LIN {X 0,Y 191.055,Z 844.267,A -85,B 0,C 180,E1 -30758.492,E2 -30758.492} C_VEL
LIN {X 0,Y 183.715,Z 843.37,A -85,B 0,C 180,E1 -30762.24,E2 -30762.24} C_VEL
LIN {X 0,Y 177.701,Z 841.067,A -85,B 0,C 180,E1 -30766.319,E2 -30766.319} C_VEL
LIN {X 0,Y 173.965,Z 838.465,A -85,B 0,C 180,E1 -30769.56,E2 -30769.56} C_VEL
LIN {X 0,Y 170.368,Z 833.668,A -85,B 0,C 180,E1 -30774.1,E2 -30774.1} C_VEL
LIN {X 0,Y 168.598,Z 829.177,A -85,B 0,C 180,E1 -30777.618,E2 -30777.618} C_VEL
LIN {X 0,Y 167.407,Z 822.526,A -85,B 0,C 180,E1 -30781.797,E2 -30781.797} C_VEL
LIN {X 0,Y 167.191,Z 815.652,A -85,B 0,C 180,E1 -30785.408,E2 -30785.408} C_VEL
LIN {X 0,Y 167.388,Z 808.865,A -85,B 0,C 180,E1 -30788.421,E2 -30788.421} C_VEL
LIN {X 0,Y 167.699,Z 800.631,A -85,B 0,C 180,E1 -30791.442,E2 -30791.442} C_VEL
LIN {X 0,Y 167.988,Z 791.47,A -85,B 0,C 180,E1 -30794.179,E2 -30794.179} C_VEL
LIN {X 0,Y 168.367,Z 782.647,A -85,B 0,C 180,E1 -30796.399,E2 -30796.399} C_VEL
LIN {X 0,Y 168.769,Z 772.895,A -85,B 0,C 180,E1 -30798.447,E2 -30798.447} C_VEL
LIN {X 0,Y 169.197,Z 762.216,A -85,B 0,C 180,E1 -30800.285,E2 -30800.285} C_VEL
LIN {X 0,Y 169.704,Z 751.249,A -85,B 0,C 180,E1 -30801.805,E2 -30801.805} C_VEL
LIN {X 0,Y 170.027,Z 740.5,A -85,B 0,C 180,E1 -30802.958,E2 -30802.958} C_VEL
LIN {X 0,Y 171.114,Z 700.591,A -85,B 0,C 180,E1 -30806.113,E2 -30806.113} C_VEL
LIN {X 0,Y 171.929,Z 668.174,A -85,B 0,C 180,E1 -30808.506,E2 -30808.506} C_VEL
LIN {X 0,Y 169.464,Z 639.672,A -85,B 0,C 180,E1 -30810.518,E2 -30810.518} C_VEL
LIN {X 0,Y 169.295,Z 636.336,A -85,B 0,C 180,E1 -30810.797,E2 -30810.797} C_VEL
LIN {X 0,Y 168.528,Z 636.419,A -85,B 0,C 180,E1 -30817.843,E2 -30817.843} C_VEL
LIN {X 0,Y 168.51,Z 636.427,A -85,B 0,C 180,E1 -30821.686,E2 -30821.686} C_VEL
LIN {X 0,Y 168.522,Z 636.419,A -85,B 0,C 180,E1 -30825.041,E2 -30825.041} C_VEL
LIN {X 0,Y 168.51,Z 636.425,A -85,B 0,C 180,E1 -30828.434,E2 -30828.434} C_VEL
LIN {X 0,Y 168.485,Z 636.43,A -85,B 0,C 180,E1 -30832.174,E2 -30832.174} C_VEL
LIN {X 0,Y 168.489,Z 636.423,A -85,B 0,C 180,E1 -30837.286,E2 -30837.286} C_VEL
LIN {X 0,Y 168.541,Z 636.422,A -85,B 0,C 180,E1 -30840.777,E2 -30840.777} C_VEL
LIN {X 0,Y 168.602,Z 636.409,A -85,B 0,C 180,E1 -30846.058,E2 -30846.058} C_VEL
LIN {X 0,Y 168.727,Z 636.397,A -85,B 0,C 180,E1 -30852.705,E2 -30852.705} C_VEL
LIN {X 0,Y 168.823,Z 636.386,A -85,B 0,C 180,E1 -30858.027,E2 -30858.027} C_VEL
LIN {X 0,Y 169.224,Z 636.335,A -85,B 0,C 180,E1 -30863.403,E2 -30863.403} C_VEL
LIN {X 0,Y 169.389,Z 636.314,A -85,B 0,C 180,E1 -30867.63,E2 -30867.63} C_VEL
LIN {X 0,Y 169.471,Z 636.309,A -85,B 0,C 180,E1 -30870,E2 -30870} C_VEL
LIN {X 0,Y 169.237,Z 636.327,A -85,B 0,C 180,E1 -30874.748,E2 -30874.748} C_VEL
LIN {X 0,Y 169.13,Z 636.346,A -85,B 0,C 180,E1 -30877.137,E2 -30877.137} C_VEL
LIN {X 0,Y 168.823,Z 636.386,A -85,B 0,C 180,E1 -30881.972,E2 -30881.972} C_VEL
LIN {X 0,Y 168.726,Z 636.397,A -85,B 0,C 180,E1 -30887.294,E2 -30887.294} C_VEL
LIN {X 0,Y 168.6,Z 636.409,A -85,B 0,C 180,E1 -30893.941,E2 -30893.941} C_VEL
LIN {X 0,Y 168.543,Z 636.422,A -85,B 0,C 180,E1 -30899.224,E2 -30899.224} C_VEL
LIN {X 0,Y 168.513,Z 636.42,A -85,B 0,C 180,E1 -30903.767,E2 -30903.767} C_VEL
LIN {X 0,Y 168.501,Z 636.428,A -85,B 0,C 180,E1 -30908.574,E2 -30908.574} C_VEL
LIN {X 0,Y 168.51,Z 636.425,A -85,B 0,C 180,E1 -30911.687,E2 -30911.687} C_VEL
LIN {X 0,Y 168.52,Z 636.42,A -85,B 0,C 180,E1 -30915.043,E2 -30915.043} C_VEL
LIN {X 0,Y 168.51,Z 636.427,A -85,B 0,C 180,E1 -30918.435,E2 -30918.435} C_VEL
LIN {X 0,Y 168.494,Z 636.423,A -85,B 0,C 180,E1 -30922.171,E2 -30922.171} C_VEL
LIN {X 0,Y 168.503,Z 636.426,A -85,B 0,C 180,E1 -30927.291,E2 -30927.291} C_VEL
LIN {X 0,Y 168.542,Z 636.414,A -85,B 0,C 180,E1 -30932.798,E2 -30932.798} C_VEL
LIN {X 0,Y 168.553,Z 636.423,A -85,B 0,C 180,E1 -30938.038,E2 -30938.038} C_VEL
LIN {X 0,Y 168.728,Z 636.39,A -85,B 0,C 180,E1 -30943.108,E2 -30943.108} C_VEL
LIN {X 0,Y 168.777,Z 636.395,A -85,B 0,C 180,E1 -30948.025,E2 -30948.025} C_VEL
LIN {X 0,Y 169.227,Z 636.329,A -85,B 0,C 180,E1 -30953.4,E2 -30953.4} C_VEL
LIN {X 0,Y 169.395,Z 636.317,A -85,B 0,C 180,E1 -30957.631,E2 -30957.631} C_VEL
LIN {X 0,Y 169.471,Z 636.305,A -85,B 0,C 180,E1 -30960.001,E2 -30960.001} C_VEL
LIN {X 0,Y 169.24,Z 636.333,A -85,B 0,C 180,E1 -30964.749,E2 -30964.749} C_VEL
LIN {X 0,Y 169.131,Z 636.349,A -85,B 0,C 180,E1 -30967.138,E2 -30967.138} C_VEL
LIN {X 0,Y 168.769,Z 636.388,A -85,B 0,C 180,E1 -30971.977,E2 -30971.977} C_VEL
LIN {X 0,Y 168.652,Z 636.408,A -85,B 0,C 180,E1 -30977.21,E2 -30977.21} C_VEL
LIN {X 0,Y 168.551,Z 636.418,A -85,B 0,C 180,E1 -30983.902,E2 -30983.902} C_VEL
LIN {X 0,Y 168.543,Z 636.42,A -85,B 0,C 180,E1 -30989.223,E2 -30989.223} C_VEL
LIN {X 0,Y 168.47,Z 636.428,A -85,B 0,C 180,E1 -30993.744,E2 -30993.744} C_VEL
LIN {X 0,Y 168.474,Z 636.429,A -85,B 0,C 180,E1 -30998.583,E2 -30998.583} C_VEL
LIN {X 0,Y 168.459,Z 636.425,A -85,B 0,C 180,E1 -31001.704,E2 -31001.704} C_VEL
LIN {X 0,Y 168.461,Z 636.432,A -85,B 0,C 180,E1 -31005.022,E2 -31005.022} C_VEL
LIN {X 0,Y 168.465,Z 636.43,A -85,B 0,C 180,E1 -31008.453,E2 -31008.453} C_VEL
LIN {X 0,Y 168.479,Z 636.425,A -85,B 0,C 180,E1 -31012.179,E2 -31012.179} C_VEL
LIN {X 0,Y 168.51,Z 636.426,A -85,B 0,C 180,E1 -31017.292,E2 -31017.292} C_VEL
LIN {X 0,Y 168.863,Z 636.379,A -85,B 0,C 180,E1 -31022.853,E2 -31022.853} C_VEL
LIN {X 0,Y 169.387,Z 636.322,A -85,B 0,C 180,E1 -31025.575,E2 -31025.575} C_VEL
LIN {X 0,Y 169.125,Z 636.516,A -85,B 0,C 180,E1 -31026.992,E2 -31026.992} C_VEL
LIN {X 0,Y 168.664,Z 639.876,A -85,B 0,C 180,E1 -31028.932,E2 -31028.932} C_VEL
LIN {X 0,Y 169.406,Z 663.952,A -85,B 0,C 180,E1 -31030.685,E2 -31030.685} C_VEL
LIN {X 0,Y 171.642,Z 691.866,A -85,B 0,C 180,E1 -31032.65,E2 -31032.65} C_VEL
LIN {X 0,Y 170.5,Z 744.148,A -85,B 0,C 180,E1 -31036.64,E2 -31036.64} C_VEL
LIN {X 0,Y 170.205,Z 756.052,A -85,B 0,C 180,E1 -31037.825,E2 -31037.825} C_VEL
LIN {X 0,Y 169.892,Z 767.351,A -85,B 0,C 180,E1 -31039.308,E2 -31039.308} C_VEL
LIN {X 0,Y 169.553,Z 776.429,A -85,B 0,C 180,E1 -31040.789,E2 -31040.789} C_VEL
LIN {X 0,Y 169.206,Z 786.88,A -85,B 0,C 180,E1 -31042.867,E2 -31042.867} C_VEL
LIN {X 0,Y 168.997,Z 795.616,A -85,B 0,C 180,E1 -31044.947,E2 -31044.947} C_VEL
LIN {X 0,Y 168.892,Z 803.11,A -85,B 0,C 180,E1 -31047.029,E2 -31047.029} C_VEL
LIN {X 0,Y 168.902,Z 810.469,A -85,B 0,C 180,E1 -31049.406,E2 -31049.406} C_VEL
LIN {X 0,Y 168.775,Z 818.031,A -85,B 0,C 180,E1 -31052.379,E2 -31052.379} C_VEL
LIN {X 0,Y 168.286,Z 825.103,A -85,B 0,C 180,E1 -31055.973,E2 -31055.973} C_VEL
LIN {X 0,Y 168,Z 830.869,A -85,B 0,C 180,E1 -31059.601,E2 -31059.601} C_VEL
LIN {X 0,Y 168.608,Z 835.707,A -85,B 0,C 180,E1 -31063.208,E2 -31063.208} C_VEL
LIN {X 0,Y 170.819,Z 840.683,A -85,B 0,C 180,E1 -31067.911,E2 -31067.911} C_VEL
LIN {X 0,Y 173.542,Z 843.594,A -85,B 0,C 180,E1 -31071.301,E2 -31071.301} C_VEL
LIN {X 0,Y 178.333,Z 846.216,A -85,B 0,C 180,E1 -31075.598,E2 -31075.598} C_VEL
LIN {X 0,Y 184.426,Z 847.512,A -85,B 0,C 180,E1 -31079.587,E2 -31079.587} C_VEL
LIN {X 0,Y 187.854,Z 847.692,A -85,B 0,C 180,E1 -31081.468,E2 -31081.468} C_VEL
LIN {X 0,Y 195.715,Z 847.111,A -85,B 0,C 180,E1 -31084.934,E2 -31084.934} C_VEL
LIN {X 0,Y 205.771,Z 844.746,A -85,B 0,C 180,E1 -31088.471,E2 -31088.471} C_VEL
LIN {X 0,Y 216.568,Z 840.579,A -85,B 0,C 180,E1 -31091.532,E2 -31091.532} C_VEL
LIN {X 0,Y 224.354,Z 836.762,A -85,B 0,C 180,E1 -31093.382,E2 -31093.382} C_VEL
LIN {X 0,Y 232.555,Z 831.917,A -85,B 0,C 180,E1 -31095.058,E2 -31095.058} C_VEL
LIN {X 0,Y 241.045,Z 825.94,A -85,B 0,C 180,E1 -31096.592,E2 -31096.592} C_VEL
LIN {X 0,Y 248.373,Z 820.093,A -85,B 0,C 180,E1 -31097.756,E2 -31097.756} C_VEL
LIN {X 0,Y 257.164,Z 811.844,A -85,B 0,C 180,E1 -31098.992,E2 -31098.992} C_VEL
LIN {X 0,Y 264.177,Z 804.216,A -85,B 0,C 180,E1 -31099.877,E2 -31099.877} C_VEL
LIN {X 0,Y 263.17,Z 805.387,A -85,B 0,C 180,E1 -31100.012,E2 -31100.012} C_VEL
LIN {X 0,Y 257.968,Z 810.774,A -85,B 0,C 180,E1 -31099.94,E2 -31099.94} C_VEL
LIN {X 0,Y 253.897,Z 814.812,A -85,B 0,C 180,E1 -31099.733,E2 -31099.733} C_VEL
LIN {X 0,Y 245.545,Z 821.967,A -85,B 0,C 180,E1 -31099.109,E2 -31099.109} C_VEL
LIN {X 0,Y 241.416,Z 825.04,A -85,B 0,C 180,E1 -31098.602,E2 -31098.602} C_VEL
LIN {X 0,Y 233.412,Z 830.545,A -85,B 0,C 180,E1 -31097.326,E2 -31097.326} C_VEL
LIN {X 0,Y 224.856,Z 835.559,A -85,B 0,C 180,E1 -31095.764,E2 -31095.764} C_VEL
LIN {X 0,Y 216.603,Z 839.644,A -85,B 0,C 180,E1 -31094.049,E2 -31094.049} C_VEL
LIN {X 0,Y 208.795,Z 842.789,A -85,B 0,C 180,E1 -31092.14,E2 -31092.14} C_VEL
LIN {X 0,Y 201.117,Z 845.175,A -85,B 0,C 180,E1 -31089.985,E2 -31089.985} C_VEL
LIN {X 0,Y 194.363,Z 846.653,A -85,B 0,C 180,E1 -31087.782,E2 -31087.782} C_VEL
LIN {X 0,Y 185.778,Z 847.498,A -85,B 0,C 180,E1 -31084.441,E2 -31084.441} C_VEL
LIN {X 0,Y 178.316,Z 847.013,A -85,B 0,C 180,E1 -31080.708,E2 -31080.708} C_VEL
LIN {X 0,Y 172.018,Z 845.234,A -85,B 0,C 180,E1 -31076.61,E2 -31076.61} C_VEL
LIN {X 0,Y 167.071,Z 842.215,A -85,B 0,C 180,E1 -31072.169,E2 -31072.169} C_VEL
LIN {X 0,Y 164.258,Z 839.064,A -85,B 0,C 180,E1 -31068.653,E2 -31068.653} C_VEL
LIN {X 0,Y 162.431,Z 835.186,A -85,B 0,C 180,E1 -31064.996,E2 -31064.996} C_VEL
LIN {X 0,Y 161.476,Z 830.456,A -85,B 0,C 180,E1 -31061.257,E2 -31061.257} C_VEL
LIN {X 0,Y 161.73,Z 822.463,A -85,B 0,C 180,E1 -31056.215,E2 -31056.215} C_VEL
LIN {X 0,Y 162.123,Z 816.783,A -85,B 0,C 180,E1 -31053.287,E2 -31053.287} C_VEL
LIN {X 0,Y 162.247,Z 808.731,A -85,B 0,C 180,E1 -31050,E2 -31050} C_VEL
LIN {X 0,Y 162.202,Z 798.946,A -85,B 0,C 180,E1 -31046.845,E2 -31046.845} C_VEL
LIN {X 0,Y 162.351,Z 789.872,A -85,B 0,C 180,E1 -31044.43,E2 -31044.43} C_VEL
LIN {X 0,Y 162.561,Z 780.372,A -85,B 0,C 180,E1 -31042.321,E2 -31042.321} C_VEL
LIN {X 0,Y 162.988,Z 769.102,A -85,B 0,C 180,E1 -31040.274,E2 -31040.274} C_VEL
LIN {X 0,Y 163.288,Z 758.249,A -85,B 0,C 180,E1 -31038.714,E2 -31038.714} C_VEL
LIN {X 0,Y 163.548,Z 746.284,A -85,B 0,C 180,E1 -31037.4,E2 -31037.4} C_VEL
LIN {X 0,Y 164.158,Z 713.491,A -85,B 0,C 180,E1 -31034.692,E2 -31034.692} C_VEL
LIN {X 0,Y 164.481,Z 689.282,A -85,B 0,C 180,E1 -31032.777,E2 -31032.777} C_VEL
LIN {X 0,Y 161.917,Z 656.305,A -85,B 0,C 180,E1 -31030.339,E2 -31030.339} C_VEL
LIN {X 0,Y 161.586,Z 639.7,A -85,B 0,C 180,E1 -31029.046,E2 -31029.046} C_VEL
LIN {X 0,Y 161.826,Z 637.261,A -85,B 0,C 180,E1 -31027.578,E2 -31027.578} C_VEL
LIN {X 0,Y 162.227,Z 637.213,A -85,B 0,C 180,E1 -31025.056,E2 -31025.056} C_VEL
LIN {X 0,Y 161.479,Z 637.299,A -85,B 0,C 180,E1 -31018.633,E2 -31018.633} C_VEL
LIN {X 0,Y 161.427,Z 637.309,A -85,B 0,C 180,E1 -31015.531,E2 -31015.531} C_VEL
LIN {X 0,Y 161.43,Z 637.299,A -85,B 0,C 180,E1 -31011.355,E2 -31011.355} C_VEL
LIN {X 0,Y 161.383,Z 637.316,A -85,B 0,C 180,E1 -31006.018,E2 -31006.018} C_VEL
LIN {X 0,Y 161.386,Z 637.306,A -85,B 0,C 180,E1 -31000.62,E2 -31000.62} C_VEL
LIN {X 0,Y 161.414,Z 637.31,A -85,B 0,C 180,E1 -30997.411,E2 -30997.411} C_VEL
LIN {X 0,Y 161.405,Z 637.312,A -85,B 0,C 180,E1 -30994.345,E2 -30994.345} C_VEL
LIN {X 0,Y 161.471,Z 637.3,A -85,B 0,C 180,E1 -30989.822,E2 -30989.822} C_VEL
LIN {X 0,Y 161.488,Z 637.301,A -85,B 0,C 180,E1 -30984.376,E2 -30984.376} C_VEL
LIN {X 0,Y 161.487,Z 637.296,A -85,B 0,C 180,E1 -30980.304,E2 -30980.304} C_VEL
LIN {X 0,Y 161.615,Z 637.283,A -85,B 0,C 180,E1 -30975.073,E2 -30975.073} C_VEL
LIN {X 0,Y 161.838,Z 637.255,A -85,B 0,C 180,E1 -30969.97,E2 -30969.97} C_VEL
LIN {X 0,Y 162.186,Z 637.214,A -85,B 0,C 180,E1 -30966.632,E2 -30966.632} C_VEL
LIN {X 0,Y 162.354,Z 637.186,A -85,B 0,C 180,E1 -30962.473,E2 -30962.473} C_VEL
LIN {X 0,Y 162.439,Z 637.181,A -85,B 0,C 180,E1 -30960.001,E2 -30960.001} C_VEL
LIN {X 0,Y 162.19,Z 637.211,A -85,B 0,C 180,E1 -30955.046,E2 -30955.046} C_VEL
LIN {X 0,Y 162.059,Z 637.222,A -85,B 0,C 180,E1 -30952.551,E2 -30952.551} C_VEL
LIN {X 0,Y 161.688,Z 637.276,A -85,B 0,C 180,E1 -30947.491,E2 -30947.491} C_VEL
LIN {X 0,Y 161.614,Z 637.277,A -85,B 0,C 180,E1 -30942.34,E2 -30942.34} C_VEL
LIN {X 0,Y 161.498,Z 637.299,A -85,B 0,C 180,E1 -30937.025,E2 -30937.025} C_VEL
LIN {X 0,Y 161.474,Z 637.301,A -85,B 0,C 180,E1 -30931.501,E2 -30931.501} C_VEL
LIN {X 0,Y 161.446,Z 637.302,A -85,B 0,C 180,E1 -30925.519,E2 -30925.519} C_VEL
LIN {X 0,Y 161.444,Z 637.304,A -85,B 0,C 180,E1 -30921.347,E2 -30921.347} C_VEL
LIN {X 0,Y 161.432,Z 637.306,A -85,B 0,C 180,E1 -30916.035,E2 -30916.035} C_VEL
LIN {X 0,Y 161.421,Z 637.308,A -85,B 0,C 180,E1 -30910.608,E2 -30910.608} C_VEL
LIN {X 0,Y 161.448,Z 637.305,A -85,B 0,C 180,E1 -30907.401,E2 -30907.401} C_VEL
LIN {X 0,Y 161.462,Z 637.298,A -85,B 0,C 180,E1 -30904.329,E2 -30904.329} C_VEL
LIN {X 0,Y 161.474,Z 637.303,A -85,B 0,C 180,E1 -30898.5,E2 -30898.5} C_VEL
LIN {X 0,Y 161.535,Z 637.29,A -85,B 0,C 180,E1 -30892.97,E2 -30892.97} C_VEL
LIN {X 0,Y 161.672,Z 637.277,A -85,B 0,C 180,E1 -30887.611,E2 -30887.611} C_VEL
LIN {X 0,Y 161.732,Z 637.267,A -85,B 0,C 180,E1 -30882.506,E2 -30882.506} C_VEL
LIN {X 0,Y 162.184,Z 637.212,A -85,B 0,C 180,E1 -30876.63,E2 -30876.63} C_VEL
LIN {X 0,Y 162.354,Z 637.19,A -85,B 0,C 180,E1 -30872.472,E2 -30872.472} C_VEL
LIN {X 0,Y 162.438,Z 637.185,A -85,B 0,C 180,E1 -30870,E2 -30870} C_VEL
LIN {X 0,Y 162.182,Z 637.206,A -85,B 0,C 180,E1 -30865.044,E2 -30865.044} C_VEL
LIN {X 0,Y 162.059,Z 637.227,A -85,B 0,C 180,E1 -30862.549,E2 -30862.549} C_VEL
LIN {X 0,Y 161.733,Z 637.267,A -85,B 0,C 180,E1 -30857.493,E2 -30857.493} C_VEL
LIN {X 0,Y 161.66,Z 637.278,A -85,B 0,C 180,E1 -30852.344,E2 -30852.344} C_VEL
LIN {X 0,Y 161.536,Z 637.29,A -85,B 0,C 180,E1 -30847.029,E2 -30847.029} C_VEL
LIN {X 0,Y 161.471,Z 637.304,A -85,B 0,C 180,E1 -30841.499,E2 -30841.499} C_VEL
LIN {X 0,Y 161.432,Z 637.307,A -85,B 0,C 180,E1 -30838.622,E2 -30838.622} C_VEL
LIN {X 0,Y 161.425,Z 637.303,A -85,B 0,C 180,E1 -30835.529,E2 -30835.529} C_VEL
LIN {X 0,Y 161.437,Z 637.307,A -85,B 0,C 180,E1 -30831.349,E2 -30831.349} C_VEL
LIN {X 0,Y 161.433,Z 637.301,A -85,B 0,C 180,E1 -30826.034,E2 -30826.034} C_VEL
LIN {X 0,Y 161.423,Z 637.309,A -85,B 0,C 180,E1 -30820.606,E2 -30820.606} C_VEL
LIN {X 0,Y 161.751,Z 637.265,A -85,B 0,C 180,E1 -30814.259,E2 -30814.259} C_VEL
LIN {X 0,Y 162.252,Z 637.213,A -85,B 0,C 180,E1 -30810.576,E2 -30810.576} C_VEL
LIN {X 0,Y 164.204,Z 662.245,A -85,B 0,C 180,E1 -30808.7,E2 -30808.7} C_VEL
LIN {X 0,Y 164.891,Z 670.706,A -85,B 0,C 180,E1 -30808.078,E2 -30808.078} C_VEL
LIN {X 0,Y 163.183,Z 736.424,A -85,B 0,C 180,E1 -30802.808,E2 -30802.808} C_VEL
LIN {X 0,Y 162.878,Z 748.151,A -85,B 0,C 180,E1 -30801.605,E2 -30801.605} C_VEL
LIN {X 0,Y 162.421,Z 759.903,A -85,B 0,C 180,E1 -30800,E2 -30800} C_VEL
LIN {X 0,Y 161.961,Z 770.643,A -85,B 0,C 180,E1 -30798.148,E2 -30798.148} C_VEL
LIN {X 0,Y 161.56,Z 781.124,A -85,B 0,C 180,E1 -30795.932,E2 -30795.932} C_VEL
LIN {X 0,Y 161.239,Z 789.408,A -85,B 0,C 180,E1 -30793.822,E2 -30793.822} C_VEL
LIN {X 0,Y 161.022,Z 797.796,A -85,B 0,C 180,E1 -30791.288,E2 -30791.288} C_VEL
LIN {X 0,Y 160.772,Z 804.868,A -85,B 0,C 180,E1 -30788.77,E2 -30788.77} C_VEL
LIN {X 0,Y 160.526,Z 812.286,A -85,B 0,C 180,E1 -30785.633,E2 -30785.633} C_VEL
LIN {X 0,Y 160.625,Z 819.692,A -85,B 0,C 180,E1 -30781.873,E2 -30781.873} C_VEL
LIN {X 0,Y 161.284,Z 824.94,A -85,B 0,C 180,E1 -30778.763,E2 -30778.763} C_VEL
LIN {X 0,Y 163.458,Z 831.717,A -85,B 0,C 180,E1 -30773.849,E2 -30773.849} C_VEL
LIN {X 0,Y 165.963,Z 835.855,A -85,B 0,C 180,E1 -30770.28,E2 -30770.28} C_VEL
LIN {X 0,Y 170.776,Z 840.005,A -85,B 0,C 180,E1 -30765.753,E2 -30765.753} C_VEL
LIN {X 0,Y 173.717,Z 841.635,A -85,B 0,C 180,E1 -30763.605,E2 -30763.605} C_VEL
LIN {X 0,Y 180.459,Z 843.787,A -85,B 0,C 180,E1 -30759.553,E2 -30759.553} C_VEL
LIN {X 0,Y 188.495,Z 844.48,A -85,B 0,C 180,E1 -30755.873,E2 -30755.873} C_VEL
LIN {X 0,Y 197.487,Z 843.746,A -85,B 0,C 180,E1 -30752.543,E2 -30752.543} C_VEL
LIN {X 0,Y 202.34,Z 842.909,A -85,B 0,C 180,E1 -30751.011,E2 -30751.011} C_VEL
LIN {X 0,Y 212.658,Z 839.96,A -85,B 0,C 180,E1 -30748.196,E2 -30748.196} C_VEL
LIN {X 0,Y 220.851,Z 836.68,A -85,B 0,C 180,E1 -30746.287,E2 -30746.287} C_VEL
LIN {X 0,Y 229.342,Z 832.371,A -85,B 0,C 180,E1 -30744.529,E2 -30744.529} C_VEL
LIN {X 0,Y 239.278,Z 826.228,A -85,B 0,C 180,E1 -30742.761,E2 -30742.761} C_VEL
LIN {X 0,Y 248.993,Z 818.86,A -85,B 0,C 180,E1 -30741.25,E2 -30741.25} C_VEL
LIN {X 0,Y 253.991,Z 814.591,A -85,B 0,C 180,E1 -30740.55,E2 -30740.55} C_VEL
LIN {X 0,Y 254.571,Z 814.072,A -85,B 0,C 180,E1 -30740.392,E2 -30740.392} C_VEL
LIN {X 0,Y 245.316,Z 822.115,A -85,B 0,C 180,E1 -30739.17,E2 -30739.17} C_VEL
LIN {X 0,Y 241.416,Z 825.04,A -85,B 0,C 180,E1 -30738.602,E2 -30738.602} C_VEL
LIN {X 0,Y 236.883,Z 828.304,A -85,B 0,C 180,E1 -30738.093,E2 -30738.093} C_VEL
LIN {X 0,Y 228.579,Z 833.287,A -85,B 0,C 180,E1 -30737.541,E2 -30737.541} C_VEL
LIN {X 0,Y 220.086,Z 837.473,A -85,B 0,C 180,E1 -30736.869,E2 -30736.869} C_VEL
LIN {X 0,Y 215.312,Z 839.46,A -85,B 0,C 180,E1 -30736.156,E2 -30736.156} C_VEL
LIN {X 0,Y 208.902,Z 842.047,A -85,B 0,C 180,E1 -30734.76,E2 -30734.76} C_VEL
LIN {X 0,Y 196.839,Z 845.42,A -85,B 0,C 180,E1 -30731.644,E2 -30731.644} C_VEL
LIN {X 0,Y 188.815,Z 846.762,A -85,B 0,C 180,E1 -30729.098,E2 -30729.098} C_VEL
LIN {X 0,Y 184.272,Z 847.179,A -85,B 0,C 180,E1 -30727.459,E2 -30727.459} C_VEL
LIN {X 0,Y 175.926,Z 846.95,A -85,B 0,C 180,E1 -30723.877,E2 -30723.877} C_VEL
LIN {X 0,Y 168.836,Z 845.452,A -85,B 0,C 180,E1 -30719.858,E2 -30719.858} C_VEL
LIN {X 0,Y 163.001,Z 842.631,A -85,B 0,C 180,E1 -30715.45,E2 -30715.45} C_VEL
LIN {X 0,Y 158.581,Z 838.543,A -85,B 0,C 180,E1 -30710.693,E2 -30710.693} C_VEL
LIN {X 0,Y 156.417,Z 834.621,A -85,B 0,C 180,E1 -30706.923,E2 -30706.923} C_VEL
LIN {X 0,Y 155.119,Z 829.85,A -85,B 0,C 180,E1 -30703.049,E2 -30703.049} C_VEL
LIN {X 0,Y 154.889,Z 823.141,A -85,B 0,C 180,E1 -30698.452,E2 -30698.452} C_VEL
LIN {X 0,Y 155.451,Z 816.467,A -85,B 0,C 180,E1 -30694.745,E2 -30694.745} C_VEL
LIN {X 0,Y 155.667,Z 810.148,A -85,B 0,C 180,E1 -30691.934,E2 -30691.934} C_VEL
LIN {X 0,Y 155.564,Z 800.186,A -85,B 0,C 180,E1 -30688.388,E2 -30688.388} C_VEL
LIN {X 0,Y 155.611,Z 790.303,A -85,B 0,C 180,E1 -30685.545,E2 -30685.545} C_VEL
LIN {X 0,Y 155.757,Z 780.676,A -85,B 0,C 180,E1 -30683.253,E2 -30683.253} C_VEL
LIN {X 0,Y 156.101,Z 770.601,A -85,B 0,C 180,E1 -30681.289,E2 -30681.289} C_VEL
LIN {X 0,Y 156.368,Z 759.098,A -85,B 0,C 180,E1 -30679.516,E2 -30679.516} C_VEL
LIN {X 0,Y 156.53,Z 748.219,A -85,B 0,C 180,E1 -30678.22,E2 -30678.22} C_VEL
LIN {X 0,Y 156.973,Z 729.692,A -85,B 0,C 180,E1 -30676.534,E2 -30676.534} C_VEL
LIN {X 0,Y 157.5,Z 689.693,A -85,B 0,C 180,E1 -30673.198,E2 -30673.198} C_VEL
LIN {X 0,Y 154.871,Z 657.033,A -85,B 0,C 180,E1 -30670.665,E2 -30670.665} C_VEL
LIN {X 0,Y 154.514,Z 639.559,A -85,B 0,C 180,E1 -30669.239,E2 -30669.239} C_VEL
LIN {X 0,Y 154.592,Z 638.16,A -85,B 0,C 180,E1 -30668.225,E2 -30668.225} C_VEL
LIN {X 0,Y 155.044,Z 638.108,A -85,B 0,C 180,E1 -30666.01,E2 -30666.01} C_VEL
LIN {X 0,Y 154.788,Z 638.132,A -85,B 0,C 180,E1 -30663.095,E2 -30663.095} C_VEL
LIN {X 0,Y 154.362,Z 638.188,A -85,B 0,C 180,E1 -30657.009,E2 -30657.009} C_VEL
LIN {X 0,Y 154.328,Z 638.191,A -85,B 0,C 180,E1 -30653.842,E2 -30653.842} C_VEL
LIN {X 0,Y 154.37,Z 638.179,A -85,B 0,C 180,E1 -30650.478,E2 -30650.478} C_VEL
LIN {X 0,Y 154.319,Z 638.194,A -85,B 0,C 180,E1 -30646.572,E2 -30646.572} C_VEL
LIN {X 0,Y 154.315,Z 638.19,A -85,B 0,C 180,E1 -30642.912,E2 -30642.912} C_VEL
LIN {X 0,Y 154.356,Z 638.187,A -85,B 0,C 180,E1 -30639.443,E2 -30639.443} C_VEL
LIN {X 0,Y 154.343,Z 638.19,A -85,B 0,C 180,E1 -30635.227,E2 -30635.227} C_VEL
LIN {X 0,Y 154.419,Z 638.178,A -85,B 0,C 180,E1 -30629.932,E2 -30629.932} C_VEL
LIN {X 0,Y 154.449,Z 638.176,A -85,B 0,C 180,E1 -30624.09,E2 -30624.09} C_VEL
LIN {X 0,Y 154.514,Z 638.172,A -85,B 0,C 180,E1 -30617.831,E2 -30617.831} C_VEL
LIN {X 0,Y 154.608,Z 638.151,A -85,B 0,C 180,E1 -30613.093,E2 -30613.093} C_VEL
LIN {X 0,Y 155.13,Z 638.093,A -85,B 0,C 180,E1 -30606.617,E2 -30606.617} C_VEL
LIN {X 0,Y 155.296,Z 638.065,A -85,B 0,C 180,E1 -30602.586,E2 -30602.586} C_VEL
LIN {X 0,Y 155.408,Z 638.057,A -85,B 0,C 180,E1 -30600.001,E2 -30600.001} C_VEL
LIN {X 0,Y 155.137,Z 638.089,A -85,B 0,C 180,E1 -30594.82,E2 -30594.82} C_VEL
LIN {X 0,Y 154.969,Z 638.105,A -85,B 0,C 180,E1 -30592.208,E2 -30592.208} C_VEL
LIN {X 0,Y 154.622,Z 638.156,A -85,B 0,C 180,E1 -30586.91,E2 -30586.91} C_VEL
LIN {X 0,Y 154.504,Z 638.168,A -85,B 0,C 180,E1 -30581.499,E2 -30581.499} C_VEL
LIN {X 0,Y 154.449,Z 638.176,A -85,B 0,C 180,E1 -30575.912,E2 -30575.912} C_VEL
LIN {X 0,Y 154.4,Z 638.184,A -85,B 0,C 180,E1 -30569.535,E2 -30569.535} C_VEL
LIN {X 0,Y 154.342,Z 638.184,A -85,B 0,C 180,E1 -30563.846,E2 -30563.846} C_VEL
LIN {X 0,Y 154.367,Z 638.187,A -85,B 0,C 180,E1 -30560.477,E2 -30560.477} C_VEL
LIN {X 0,Y 154.37,Z 638.187,A -85,B 0,C 180,E1 -30556.551,E2 -30556.551} C_VEL
LIN {X 0,Y 154.366,Z 638.181,A -85,B 0,C 180,E1 -30552.893,E2 -30552.893} C_VEL
LIN {X 0,Y 154.39,Z 638.186,A -85,B 0,C 180,E1 -30549.431,E2 -30549.431} C_VEL
LIN {X 0,Y 154.397,Z 638.178,A -85,B 0,C 180,E1 -30545.256,E2 -30545.256} C_VEL
LIN {X 0,Y 154.426,Z 638.183,A -85,B 0,C 180,E1 -30539.929,E2 -30539.929} C_VEL
LIN {X 0,Y 154.489,Z 638.166,A -85,B 0,C 180,E1 -30534.082,E2 -30534.082} C_VEL
LIN {X 0,Y 154.605,Z 638.158,A -85,B 0,C 180,E1 -30527.938,E2 -30527.938} C_VEL
LIN {X 0,Y 154.66,Z 638.147,A -85,B 0,C 180,E1 -30523.087,E2 -30523.087} C_VEL
LIN {X 0,Y 155.127,Z 638.091,A -85,B 0,C 180,E1 -30516.615,E2 -30516.615} C_VEL
LIN {X 0,Y 155.296,Z 638.069,A -85,B 0,C 180,E1 -30512.585,E2 -30512.585} C_VEL
LIN {X 0,Y 155.407,Z 638.061,A -85,B 0,C 180,E1 -30510,E2 -30510} C_VEL
LIN {X 0,Y 155.129,Z 638.084,A -85,B 0,C 180,E1 -30504.818,E2 -30504.818} C_VEL
LIN {X 0,Y 154.97,Z 638.112,A -85,B 0,C 180,E1 -30502.206,E2 -30502.206} C_VEL
LIN {X 0,Y 154.661,Z 638.147,A -85,B 0,C 180,E1 -30496.912,E2 -30496.912} C_VEL
LIN {X 0,Y 154.554,Z 638.165,A -85,B 0,C 180,E1 -30491.503,E2 -30491.503} C_VEL
LIN {X 0,Y 154.455,Z 638.17,A -85,B 0,C 180,E1 -30485.09,E2 -30485.09} C_VEL
LIN {X 0,Y 154.394,Z 638.184,A -85,B 0,C 180,E1 -30479.537,E2 -30479.537} C_VEL
LIN {X 0,Y 154.329,Z 638.19,A -85,B 0,C 180,E1 -30473.841,E2 -30473.841} C_VEL
LIN {X 0,Y 154.368,Z 638.189,A -85,B 0,C 180,E1 -30470.476,E2 -30470.476} C_VEL
LIN {X 0,Y 154.371,Z 638.181,A -85,B 0,C 180,E1 -30466.549,E2 -30466.549} C_VEL
LIN {X 0,Y 154.367,Z 638.187,A -85,B 0,C 180,E1 -30462.891,E2 -30462.891} C_VEL
LIN {X 0,Y 154.393,Z 638.183,A -85,B 0,C 180,E1 -30459.43,E2 -30459.43} C_VEL
LIN {X 0,Y 154.878,Z 638.123,A -85,B 0,C 180,E1 -30452.867,E2 -30452.867} C_VEL
LIN {X 0,Y 155.22,Z 638.089,A -85,B 0,C 180,E1 -30450.309,E2 -30450.309} C_VEL
LIN {X 0,Y 157.44,Z 664.609,A -85,B 0,C 180,E1 -30448.235,E2 -30448.235} C_VEL
LIN {X 0,Y 157.822,Z 671.244,A -85,B 0,C 180,E1 -30447.719,E2 -30447.719} C_VEL
LIN {X 0,Y 156.257,Z 735.722,A -85,B 0,C 180,E1 -30442.309,E2 -30442.309} C_VEL
LIN {X 0,Y 155.945,Z 749.039,A -85,B 0,C 180,E1 -30440.868,E2 -30440.868} C_VEL
LIN {X 0,Y 155.475,Z 759.899,A -85,B 0,C 180,E1 -30439.302,E2 -30439.302} C_VEL
LIN {X 0,Y 155.095,Z 770.423,A -85,B 0,C 180,E1 -30437.385,E2 -30437.385} C_VEL
LIN {X 0,Y 154.802,Z 779.378,A -85,B 0,C 180,E1 -30435.415,E2 -30435.415} C_VEL
LIN {X 0,Y 154.503,Z 789.371,A -85,B 0,C 180,E1 -30432.767,E2 -30432.767} C_VEL
LIN {X 0,Y 154.308,Z 796.764,A -85,B 0,C 180,E1 -30430.46,E2 -30430.46} C_VEL
LIN {X 0,Y 154.049,Z 805.511,A -85,B 0,C 180,E1 -30427.182,E2 -30427.182} C_VEL
LIN {X 0,Y 153.849,Z 812.762,A -85,B 0,C 180,E1 -30423.915,E2 -30423.915} C_VEL
LIN {X 0,Y 154.249,Z 819.956,A -85,B 0,C 180,E1 -30419.999,E2 -30419.999} C_VEL
LIN {X 0,Y 155.406,Z 826.048,A -85,B 0,C 180,E1 -30416.123,E2 -30416.123} C_VEL
LIN {X 0,Y 157.337,Z 831.193,A -85,B 0,C 180,E1 -30412.324,E2 -30412.324} C_VEL
LIN {X 0,Y 161.291,Z 836.545,A -85,B 0,C 180,E1 -30407.458,E2 -30407.458} C_VEL
LIN {X 0,Y 163.908,Z 838.772,A -85,B 0,C 180,E1 -30405.142,E2 -30405.142} C_VEL
LIN {X 0,Y 170.115,Z 842.173,A -85,B 0,C 180,E1 -30400.767,E2 -30400.767} C_VEL
LIN {X 0,Y 177.68,Z 844.122,A -85,B 0,C 180,E1 -30396.782,E2 -30396.782} C_VEL
LIN {X 0,Y 186.389,Z 844.686,A -85,B 0,C 180,E1 -30393.194,E2 -30393.194} C_VEL
LIN {X 0,Y 191.405,Z 844.477,A -85,B 0,C 180,E1 -30391.436,E2 -30391.436} C_VEL
LIN {X 0,Y 201.172,Z 842.999,A -85,B 0,C 180,E1 -30388.515,E2 -30388.515} C_VEL
LIN {X 0,Y 212.072,Z 839.844,A -85,B 0,C 180,E1 -30385.841,E2 -30385.841} C_VEL
LIN {X 0,Y 220.651,Z 836.483,A -85,B 0,C 180,E1 -30384.036,E2 -30384.036} C_VEL
LIN {X 0,Y 230.336,Z 831.646,A -85,B 0,C 180,E1 -30382.247,E2 -30382.247} C_VEL
LIN {X 0,Y 239.654,Z 825.897,A -85,B 0,C 180,E1 -30380.77,E2 -30380.77} C_VEL
LIN {X 0,Y 240.313,Z 825.446,A -85,B 0,C 180,E1 -30380.343,E2 -30380.343} C_VEL
LIN {X 0,Y 231.717,Z 831.103,A -85,B 0,C 180,E1 -30379.088,E2 -30379.088} C_VEL
LIN {X 0,Y 222.897,Z 835.971,A -85,B 0,C 180,E1 -30377.602,E2 -30377.602} C_VEL
LIN {X 0,Y 215.312,Z 839.46,A -85,B 0,C 180,E1 -30376.156,E2 -30376.156} C_VEL
LIN {X 0,Y 210.472,Z 841.384,A -85,B 0,C 180,E1 -30375.371,E2 -30375.371} C_VEL
LIN {X 0,Y 199.839,Z 844.436,A -85,B 0,C 180,E1 -30374.137,E2 -30374.137} C_VEL
LIN {X 0,Y 192.892,Z 845.699,A -85,B 0,C 180,E1 -30373.141,E2 -30373.141} C_VEL
LIN {X 0,Y 188.301,Z 846.385,A -85,B 0,C 180,E1 -30372.075,E2 -30372.075} C_VEL
LIN {X 0,Y 178.709,Z 846.954,A -85,B 0,C 180,E1 -30368.838,E2 -30368.838} C_VEL
LIN {X 0,Y 170.107,Z 846.237,A -85,B 0,C 180,E1 -30365.203,E2 -30365.203} C_VEL
LIN {X 0,Y 166.357,Z 845.5,A -85,B 0,C 180,E1 -30363.187,E2 -30363.187} C_VEL
LIN {X 0,Y 159.637,Z 843.013,A -85,B 0,C 180,E1 -30358.859,E2 -30358.859} C_VEL
LIN {X 0,Y 154.314,Z 839.17,A -85,B 0,C 180,E1 -30354.112,E2 -30354.112} C_VEL
LIN {X 0,Y 150.597,Z 834.003,A -85,B 0,C 180,E1 -30349.001,E2 -30349.001} C_VEL
LIN {X 0,Y 148.962,Z 829.232,A -85,B 0,C 180,E1 -30344.989,E2 -30344.989} C_VEL
LIN {X 0,Y 148.384,Z 822.448,A -85,B 0,C 180,E1 -30340.197,E2 -30340.197} C_VEL
LIN {X 0,Y 148.844,Z 815.499,A -85,B 0,C 180,E1 -30336.056,E2 -30336.056} C_VEL
LIN {X 0,Y 149.13,Z 808.259,A -85,B 0,C 180,E1 -30332.693,E2 -30332.693} C_VEL
LIN {X 0,Y 149.003,Z 798.966,A -85,B 0,C 180,E1 -30329.327,E2 -30329.327} C_VEL
LIN {X 0,Y 149.006,Z 788.702,A -85,B 0,C 180,E1 -30326.295,E2 -30326.295} C_VEL
LIN {X 0,Y 149.107,Z 778.954,A -85,B 0,C 180,E1 -30323.922,E2 -30323.922} C_VEL
LIN {X 0,Y 149.36,Z 768.988,A -85,B 0,C 180,E1 -30321.913,E2 -30321.913} C_VEL
LIN {X 0,Y 149.574,Z 757.837,A -85,B 0,C 180,E1 -30320.123,E2 -30320.123} C_VEL
LIN {X 0,Y 149.729,Z 746.29,A -85,B 0,C 180,E1 -30318.704,E2 -30318.704} C_VEL
LIN {X 0,Y 150.174,Z 719.804,A -85,B 0,C 180,E1 -30316.257,E2 -30316.257} C_VEL
LIN {X 0,Y 150.539,Z 690.129,A -85,B 0,C 180,E1 -30313.659,E2 -30313.659} C_VEL
LIN {X 0,Y 147.828,Z 657.031,A -85,B 0,C 180,E1 -30310.979,E2 -30310.979} C_VEL
LIN {X 0,Y 147.435,Z 639.312,A -85,B 0,C 180,E1 -30309.399,E2 -30309.399} C_VEL
LIN {X 0,Y 147.424,Z 639.054,A -85,B 0,C 180,E1 -30309.125,E2 -30309.125} C_VEL
LIN {X 0,Y 148.025,Z 638.981,A -85,B 0,C 180,E1 -30304.795,E2 -30304.795} C_VEL
LIN {X 0,Y 147.369,Z 639.057,A -85,B 0,C 180,E1 -30298.478,E2 -30298.478} C_VEL
LIN {X 0,Y 147.287,Z 639.069,A -85,B 0,C 180,E1 -30293.947,E2 -30293.947} C_VEL
LIN {X 0,Y 147.242,Z 639.074,A -85,B 0,C 180,E1 -30288.242,E2 -30288.242} C_VEL
LIN {X 0,Y 147.24,Z 639.076,A -85,B 0,C 180,E1 -30284.474,E2 -30284.474} C_VEL
LIN {X 0,Y 147.269,Z 639.065,A -85,B 0,C 180,E1 -30280.449,E2 -30280.449} C_VEL
LIN {X 0,Y 147.276,Z 639.07,A -85,B 0,C 180,E1 -30274.801,E2 -30274.801} C_VEL
LIN {X 0,Y 147.3,Z 639.061,A -85,B 0,C 180,E1 -30271.137,E2 -30271.137} C_VEL
LIN {X 0,Y 147.358,Z 639.06,A -85,B 0,C 180,E1 -30265.329,E2 -30265.329} C_VEL
LIN {X 0,Y 147.388,Z 639.056,A -85,B 0,C 180,E1 -30259.432,E2 -30259.432} C_VEL
LIN {X 0,Y 147.533,Z 639.034,A -85,B 0,C 180,E1 -30253.733,E2 -30253.733} C_VEL
LIN {X 0,Y 148.077,Z 638.972,A -85,B 0,C 180,E1 -30246.61,E2 -30246.61} C_VEL
LIN {X 0,Y 148.24,Z 638.944,A -85,B 0,C 180,E1 -30242.709,E2 -30242.709} C_VEL
LIN {X 0,Y 148.377,Z 638.932,A -85,B 0,C 180,E1 -30240.001,E2 -30240.001} C_VEL
LIN {X 0,Y 148.085,Z 638.968,A -85,B 0,C 180,E1 -30234.573,E2 -30234.573} C_VEL
LIN {X 0,Y 147.89,Z 638.988,A -85,B 0,C 180,E1 -30231.832,E2 -30231.832} C_VEL
LIN {X 0,Y 147.55,Z 639.038,A -85,B 0,C 180,E1 -30226.27,E2 -30226.27} C_VEL
LIN {X 0,Y 147.488,Z 639.039,A -85,B 0,C 180,E1 -30221.773,E2 -30221.773} C_VEL
LIN {X 0,Y 147.379,Z 639.059,A -85,B 0,C 180,E1 -30217.654,E2 -30217.654} C_VEL
LIN {X 0,Y 147.368,Z 639.056,A -85,B 0,C 180,E1 -30214.564,E2 -30214.564} C_VEL
LIN {X 0,Y 147.305,Z 639.068,A -85,B 0,C 180,E1 -30208.464,E2 -30208.464} C_VEL
LIN {X 0,Y 147.3,Z 639.061,A -85,B 0,C 180,E1 -30203.938,E2 -30203.938} C_VEL
LIN {X 0,Y 147.271,Z 639.073,A -85,B 0,C 180,E1 -30198.253,E2 -30198.253} C_VEL
LIN {X 0,Y 147.302,Z 639.062,A -85,B 0,C 180,E1 -30194.5,E2 -30194.5} C_VEL
LIN {X 0,Y 147.299,Z 639.07,A -85,B 0,C 180,E1 -30188.183,E2 -30188.183} C_VEL
LIN {X 0,Y 147.327,Z 639.059,A -85,B 0,C 180,E1 -30184.786,E2 -30184.786} C_VEL
LIN {X 0,Y 147.34,Z 639.062,A -85,B 0,C 180,E1 -30181.164,E2 -30181.164} C_VEL
LIN {X 0,Y 147.378,Z 639.052,A -85,B 0,C 180,E1 -30175.324,E2 -30175.324} C_VEL
LIN {X 0,Y 147.451,Z 639.05,A -85,B 0,C 180,E1 -30169.422,E2 -30169.422} C_VEL
LIN {X 0,Y 147.547,Z 639.036,A -85,B 0,C 180,E1 -30166.549,E2 -30166.549} C_VEL
LIN {X 0,Y 147.687,Z 639.019,A -85,B 0,C 180,E1 -30160.935,E2 -30160.935} C_VEL
LIN {X 0,Y 148.078,Z 638.963,A -85,B 0,C 180,E1 -30155.428,E2 -30155.428} C_VEL
LIN {X 0,Y 148.376,Z 638.937,A -85,B 0,C 180,E1 -30149.999,E2 -30149.999} C_VEL
LIN {X 0,Y 148.078,Z 638.963,A -85,B 0,C 180,E1 -30144.571,E2 -30144.571} C_VEL
LIN {X 0,Y 147.687,Z 639.019,A -85,B 0,C 180,E1 -30139.064,E2 -30139.064} C_VEL
LIN {X 0,Y 147.547,Z 639.036,A -85,B 0,C 180,E1 -30133.45,E2 -30133.45} C_VEL
LIN {X 0,Y 147.412,Z 639.05,A -85,B 0,C 180,E1 -30127.658,E2 -30127.658} C_VEL
LIN {X 0,Y 147.37,Z 639.053,A -85,B 0,C 180,E1 -30124.561,E2 -30124.561} C_VEL
LIN {X 0,Y 147.28,Z 639.07,A -85,B 0,C 180,E1 -30118.456,E2 -30118.456} C_VEL
LIN {X 0,Y 147.287,Z 639.067,A -85,B 0,C 180,E1 -30113.944,E2 -30113.944} C_VEL
LIN {X 0,Y 147.272,Z 639.069,A -85,B 0,C 180,E1 -30108.251,E2 -30108.251} C_VEL
LIN {X 0,Y 147.304,Z 639.063,A -85,B 0,C 180,E1 -30104.498,E2 -30104.498} C_VEL
LIN {X 0,Y 147.358,Z 639.057,A -85,B 0,C 180,E1 -30098.164,E2 -30098.164} C_VEL
LIN {X 0,Y 148.167,Z 638.967,A -85,B 0,C 180,E1 -30090.542,E2 -30090.542} C_VEL
LIN {X 0,Y 148.227,Z 638.959,A -85,B 0,C 180,E1 -30089.989,E2 -30089.989} C_VEL
LIN {X 0,Y 150.374,Z 664.663,A -85,B 0,C 180,E1 -30087.907,E2 -30087.907} C_VEL
LIN {X 0,Y 150.81,Z 670.632,A -85,B 0,C 180,E1 -30087.426,E2 -30087.426} C_VEL
LIN {X 0,Y 149.438,Z 734.013,A -85,B 0,C 180,E1 -30081.823,E2 -30081.823} C_VEL
LIN {X 0,Y 149.107,Z 748.527,A -85,B 0,C 180,E1 -30080.193,E2 -30080.193} C_VEL
LIN {X 0,Y 148.676,Z 759.435,A -85,B 0,C 180,E1 -30078.533,E2 -30078.533} C_VEL
LIN {X 0,Y 148.317,Z 770.328,A -85,B 0,C 180,E1 -30076.46,E2 -30076.46} C_VEL
LIN {X 0,Y 148.053,Z 780.728,A -85,B 0,C 180,E1 -30074.031,E2 -30074.031} C_VEL
LIN {X 0,Y 147.814,Z 789.32,A -85,B 0,C 180,E1 -30071.618,E2 -30071.618} C_VEL
LIN {X 0,Y 147.582,Z 797.565,A -85,B 0,C 180,E1 -30068.872,E2 -30068.872} C_VEL
LIN {X 0,Y 147.41,Z 804.539,A -85,B 0,C 180,E1 -30066.136,E2 -30066.136} C_VEL
LIN {X 0,Y 147.331,Z 812.993,A -85,B 0,C 180,E1 -30062.043,E2 -30062.043} C_VEL
LIN {X 0,Y 147.962,Z 819.885,A -85,B 0,C 180,E1 -30058.137,E2 -30058.137} C_VEL
LIN {X 0,Y 149.151,Z 825.326,A -85,B 0,C 180,E1 -30054.61,E2 -30054.61} C_VEL
LIN {X 0,Y 152.289,Z 831.964,A -85,B 0,C 180,E1 -30049.398,E2 -30049.398} C_VEL
LIN {X 0,Y 155.704,Z 836.094,A -85,B 0,C 180,E1 -30045.674,E2 -30045.674} C_VEL
LIN {X 0,Y 160.104,Z 839.443,A -85,B 0,C 180,E1 -30042.166,E2 -30042.166} C_VEL
LIN {X 0,Y 167.051,Z 842.606,A -85,B 0,C 180,E1 -30037.829,E2 -30037.829} C_VEL
LIN {X 0,Y 175.347,Z 844.435,A -85,B 0,C 180,E1 -30033.933,E2 -30033.933} C_VEL
LIN {X 0,Y 184.752,Z 844.901,A -85,B 0,C 180,E1 -30030.47,E2 -30030.47} C_VEL
LIN {X 0,Y 189.773,Z 844.706,A -85,B 0,C 180,E1 -30028.886,E2 -30028.886} C_VEL
LIN {X 0,Y 200.481,Z 843.038,A -85,B 0,C 180,E1 -30026.012,E2 -30026.012} C_VEL
LIN {X 0,Y 211.866,Z 839.82,A -85,B 0,C 180,E1 -30023.48,E2 -30023.48} C_VEL
LIN {X 0,Y 220.836,Z 836.359,A -85,B 0,C 180,E1 -30021.793,E2 -30021.793} C_VEL
LIN {X 0,Y 225.234,Z 834.308,A -85,B 0,C 180,E1 -30021.03,E2 -30021.03} C_VEL
LIN {X 0,Y 227.211,Z 833.409,A -85,B 0,C 180,E1 -30020.417,E2 -30020.417} C_VEL
LIN {X 0,Y 218.237,Z 837.832,A -85,B 0,C 180,E1 -30018.96,E2 -30018.96} C_VEL
LIN {X 0,Y 209.518,Z 841.273,A -85,B 0,C 180,E1 -30017.349,E2 -30017.349} C_VEL
LIN {X 0,Y 198.53,Z 844.533,A -85,B 0,C 180,E1 -30014.881,E2 -30014.881} C_VEL
LIN {X 0,Y 188.301,Z 846.385,A -85,B 0,C 180,E1 -30012.075,E2 -30012.075} C_VEL
LIN {X 0,Y 183.722,Z 846.842,A -85,B 0,C 180,E1 -30010.93,E2 -30010.93} C_VEL
LIN {X 0,Y 175.176,Z 846.768,A -85,B 0,C 180,E1 -30009.31,E2 -30009.31} C_VEL
LIN {X 0,Y 168.53,Z 846.168,A -85,B 0,C 180,E1 -30007.888,E2 -30007.888} C_VEL
LIN {X 0,Y 164.283,Z 845.446,A -85,B 0,C 180,E1 -30006.508,E2 -30006.508} C_VEL
LIN {X 0,Y 163.123,Z 845.147,A -85,B 0,C 180,E1 -30005.963,E2 -30005.963} C_VEL
LIN {X 0,Y 156.87,Z 843.157,A -85,B 0,C 180,E1 -30002.4,E2 -30002.4} C_VEL
LIN {X 0,Y 149.845,Z 839.061,A -85,B 0,C 180,E1 -29996.992,E2 -29996.992} C_VEL
LIN {X 0,Y 145.875,Z 834.768,A -85,B 0,C 180,E1 -29992.591,E2 -29992.591} C_VEL
LIN {X 0,Y 143.019,Z 828.521,A -85,B 0,C 180,E1 -29987.089,E2 -29987.089} C_VEL
LIN {X 0,Y 142.012,Z 821.747,A -85,B 0,C 180,E1 -29982.101,E2 -29982.101} C_VEL
LIN {X 0,Y 142.381,Z 814.128,A -85,B 0,C 180,E1 -29977.386,E2 -29977.386} C_VEL
LIN {X 0,Y 142.648,Z 807.848,A -85,B 0,C 180,E1 -29974.224,E2 -29974.224} C_VEL
LIN {X 0,Y 142.523,Z 799.88,A -85,B 0,C 180,E1 -29971.057,E2 -29971.057} C_VEL
LIN {X 0,Y 142.425,Z 788.633,A -85,B 0,C 180,E1 -29967.534,E2 -29967.534} C_VEL
LIN {X 0,Y 142.457,Z 779.014,A -85,B 0,C 180,E1 -29965.064,E2 -29965.064} C_VEL
LIN {X 0,Y 142.673,Z 769.115,A -85,B 0,C 180,E1 -29962.951,E2 -29962.951} C_VEL
LIN {X 0,Y 142.83,Z 757.612,A -85,B 0,C 180,E1 -29961.007,E2 -29961.007} C_VEL
LIN {X 0,Y 142.929,Z 746.203,A -85,B 0,C 180,E1 -29959.534,E2 -29959.534} C_VEL
LIN {X 0,Y 143.289,Z 719.891,A -85,B 0,C 180,E1 -29956.935,E2 -29956.935} C_VEL
LIN {X 0,Y 143.475,Z 689.555,A -85,B 0,C 180,E1 -29954.107,E2 -29954.107} C_VEL
LIN {X 0,Y 140.806,Z 656.382,A -85,B 0,C 180,E1 -29951.296,E2 -29951.296} C_VEL
LIN {X 0,Y 140.413,Z 639.924,A -85,B 0,C 180,E1 -29949.795,E2 -29949.795} C_VEL
LIN {X 0,Y 140.723,Z 639.891,A -85,B 0,C 180,E1 -29946.535,E2 -29946.535} C_VEL
LIN {X 0,Y 140.731,Z 639.884,A -85,B 0,C 180,E1 -29943.389,E2 -29943.389} C_VEL
LIN {X 0,Y 140.225,Z 639.949,A -85,B 0,C 180,E1 -29936.67,E2 -29936.67} C_VEL
LIN {X 0,Y 140.2,Z 639.949,A -85,B 0,C 180,E1 -29933.07,E2 -29933.07} C_VEL
LIN {X 0,Y 140.221,Z 639.947,A -85,B 0,C 180,E1 -29928.53,E2 -29928.53} C_VEL
LIN {X 0,Y 140.196,Z 639.954,A -85,B 0,C 180,E1 -29924.385,E2 -29924.385} C_VEL
LIN {X 0,Y 140.221,Z 639.942,A -85,B 0,C 180,E1 -29920.496,E2 -29920.496} C_VEL
LIN {X 0,Y 140.23,Z 639.949,A -85,B 0,C 180,E1 -29916.827,E2 -29916.827} C_VEL
LIN {X 0,Y 140.222,Z 639.942,A -85,B 0,C 180,E1 -29911.877,E2 -29911.877} C_VEL
LIN {X 0,Y 140.29,Z 639.943,A -85,B 0,C 180,E1 -29906.012,E2 -29906.012} C_VEL
LIN {X 0,Y 140.389,Z 639.928,A -85,B 0,C 180,E1 -29898.565,E2 -29898.565} C_VEL
LIN {X 0,Y 140.44,Z 639.922,A -85,B 0,C 180,E1 -29894.441,E2 -29894.441} C_VEL
LIN {X 0,Y 140.786,Z 639.879,A -85,B 0,C 180,E1 -29888.585,E2 -29888.585} C_VEL
LIN {X 0,Y 141.041,Z 639.847,A -85,B 0,C 180,E1 -29885.701,E2 -29885.701} C_VEL
LIN {X 0,Y 141.346,Z 639.808,A -85,B 0,C 180,E1 -29880.001,E2 -29880.001} C_VEL
LIN {X 0,Y 141.041,Z 639.844,A -85,B 0,C 180,E1 -29874.301,E2 -29874.301} C_VEL
LIN {X 0,Y 140.569,Z 639.907,A -85,B 0,C 180,E1 -29868.504,E2 -29868.504} C_VEL
LIN {X 0,Y 140.461,Z 639.911,A -85,B 0,C 180,E1 -29862.591,E2 -29862.591} C_VEL
LIN {X 0,Y 140.285,Z 639.942,A -85,B 0,C 180,E1 -29856.458,E2 -29856.458} C_VEL
LIN {X 0,Y 140.268,Z 639.935,A -85,B 0,C 180,E1 -29853.294,E2 -29853.294} C_VEL
LIN {X 0,Y 140.24,Z 639.95,A -85,B 0,C 180,E1 -29848.111,E2 -29848.111} C_VEL
LIN {X 0,Y 140.24,Z 639.94,A -85,B 0,C 180,E1 -29843.047,E2 -29843.047} C_VEL
LIN {X 0,Y 140.242,Z 639.948,A -85,B 0,C 180,E1 -29838.519,E2 -29838.519} C_VEL
LIN {X 0,Y 140.273,Z 639.937,A -85,B 0,C 180,E1 -29834.353,E2 -29834.353} C_VEL
LIN {X 0,Y 140.236,Z 639.947,A -85,B 0,C 180,E1 -29830.49,E2 -29830.49} C_VEL
LIN {X 0,Y 140.254,Z 639.945,A -85,B 0,C 180,E1 -29826.819,E2 -29826.819} C_VEL
LIN {X 0,Y 140.283,Z 639.939,A -85,B 0,C 180,E1 -29821.918,E2 -29821.918} C_VEL
LIN {X 0,Y 140.302,Z 639.936,A -85,B 0,C 180,E1 -29816.024,E2 -29816.024} C_VEL
LIN {X 0,Y 140.357,Z 639.933,A -85,B 0,C 180,E1 -29810.446,E2 -29810.446} C_VEL
LIN {X 0,Y 140.494,Z 639.914,A -85,B 0,C 180,E1 -29807.405,E2 -29807.405} C_VEL
LIN {X 0,Y 140.591,Z 639.904,A -85,B 0,C 180,E1 -29801.495,E2 -29801.495} C_VEL
LIN {X 0,Y 141.039,Z 639.84,A -85,B 0,C 180,E1 -29795.7,E2 -29795.7} C_VEL
LIN {X 0,Y 141.345,Z 639.812,A -85,B 0,C 180,E1 -29789.999,E2 -29789.999} C_VEL
LIN {X 0,Y 141.039,Z 639.84,A -85,B 0,C 180,E1 -29784.299,E2 -29784.299} C_VEL
LIN {X 0,Y 140.592,Z 639.904,A -85,B 0,C 180,E1 -29778.504,E2 -29778.504} C_VEL
LIN {X 0,Y 140.495,Z 639.914,A -85,B 0,C 180,E1 -29772.594,E2 -29772.594} C_VEL
LIN {X 0,Y 140.306,Z 639.933,A -85,B 0,C 180,E1 -29766.46,E2 -29766.46} C_VEL
LIN {X 0,Y 140.27,Z 639.942,A -85,B 0,C 180,E1 -29763.293,E2 -29763.293} C_VEL
LIN {X 0,Y 140.22,Z 639.947,A -85,B 0,C 180,E1 -29758.123,E2 -29758.123} C_VEL
LIN {X 0,Y 140.202,Z 639.951,A -85,B 0,C 180,E1 -29753.067,E2 -29753.067} C_VEL
LIN {X 0,Y 140.243,Z 639.946,A -85,B 0,C 180,E1 -29748.517,E2 -29748.517} C_VEL
LIN {X 0,Y 140.274,Z 639.939,A -85,B 0,C 180,E1 -29744.351,E2 -29744.351} C_VEL
LIN {X 0,Y 140.239,Z 639.948,A -85,B 0,C 180,E1 -29740.488,E2 -29740.488} C_VEL
LIN {X 0,Y 140.697,Z 639.89,A -85,B 0,C 180,E1 -29733.203,E2 -29733.203} C_VEL
LIN {X 0,Y 141.222,Z 639.831,A -85,B 0,C 180,E1 -29729.671,E2 -29729.671} C_VEL
LIN {X 0,Y 143.423,Z 665.53,A -85,B 0,C 180,E1 -29727.451,E2 -29727.451} C_VEL
LIN {X 0,Y 143.727,Z 671.842,A -85,B 0,C 180,E1 -29726.908,E2 -29726.908} C_VEL
LIN {X 0,Y 142.597,Z 733.525,A -85,B 0,C 180,E1 -29721.096,E2 -29721.096} C_VEL
LIN {X 0,Y 142.283,Z 748.919,A -85,B 0,C 180,E1 -29719.285,E2 -29719.285} C_VEL
LIN {X 0,Y 141.843,Z 759.758,A -85,B 0,C 180,E1 -29717.534,E2 -29717.534} C_VEL
LIN {X 0,Y 141.572,Z 770.336,A -85,B 0,C 180,E1 -29715.421,E2 -29715.421} C_VEL
LIN {X 0,Y 141.373,Z 779.359,A -85,B 0,C 180,E1 -29713.246,E2 -29713.246} C_VEL
LIN {X 0,Y 141.184,Z 789.225,A -85,B 0,C 180,E1 -29710.36,E2 -29710.36} C_VEL
LIN {X 0,Y 141.011,Z 798.164,A -85,B 0,C 180,E1 -29707.131,E2 -29707.131} C_VEL
LIN {X 0,Y 140.865,Z 804.86,A -85,B 0,C 180,E1 -29704.277,E2 -29704.277} C_VEL
LIN {X 0,Y 140.986,Z 813.22,A -85,B 0,C 180,E1 -29699.999,E2 -29699.999} C_VEL
LIN {X 0,Y 141.957,Z 820.295,A -85,B 0,C 180,E1 -29695.755,E2 -29695.755} C_VEL
LIN {X 0,Y 143.819,Z 826.235,A -85,B 0,C 180,E1 -29691.598,E2 -29691.598} C_VEL
LIN {X 0,Y 146.533,Z 831.291,A -85,B 0,C 180,E1 -29687.577,E2 -29687.577} C_VEL
LIN {X 0,Y 151.806,Z 836.729,A -85,B 0,C 180,E1 -29682.547,E2 -29682.547} C_VEL
LIN {X 0,Y 156.717,Z 839.951,A -85,B 0,C 180,E1 -29679.049,E2 -29679.049} C_VEL
LIN {X 0,Y 164.526,Z 843.015,A -85,B 0,C 180,E1 -29674.802,E2 -29674.802} C_VEL
LIN {X 0,Y 173.542,Z 844.738,A -85,B 0,C 180,E1 -29671.03,E2 -29671.03} C_VEL
LIN {X 0,Y 180.369,Z 845.235,A -85,B 0,C 180,E1 -29668.688,E2 -29668.688} C_VEL
LIN {X 0,Y 188.889,Z 844.894,A -85,B 0,C 180,E1 -29666.204,E2 -29666.204} C_VEL
LIN {X 0,Y 200.706,Z 842.996,A -85,B 0,C 180,E1 -29663.387,E2 -29663.387} C_VEL
LIN {X 0,Y 212.109,Z 839.796,A -85,B 0,C 180,E1 -29661.138,E2 -29661.138} C_VEL
LIN {X 0,Y 214.133,Z 839.086,A -85,B 0,C 180,E1 -29660.785,E2 -29660.785} C_VEL
LIN {X 0,Y 213.478,Z 839.358,A -85,B 0,C 180,E1 -29660.358,E2 -29660.358} C_VEL
LIN {X 0,Y 204.805,Z 842.33,A -85,B 0,C 180,E1 -29658.8,E2 -29658.8} C_VEL
LIN {X 0,Y 199.115,Z 843.944,A -85,B 0,C 180,E1 -29657.624,E2 -29657.624} C_VEL
LIN {X 0,Y 188.184,Z 846.004,A -85,B 0,C 180,E1 -29655.009,E2 -29655.009} C_VEL
LIN {X 0,Y 178.041,Z 846.749,A -85,B 0,C 180,E1 -29651.976,E2 -29651.976} C_VEL
LIN {X 0,Y 168.686,Z 846.215,A -85,B 0,C 180,E1 -29648.526,E2 -29648.526} C_VEL
LIN {X 0,Y 163.123,Z 845.147,A -85,B 0,C 180,E1 -29645.963,E2 -29645.963} C_VEL
LIN {X 0,Y 159.455,Z 844.183,A -85,B 0,C 180,E1 -29644.364,E2 -29644.364} C_VEL
LIN {X 0,Y 153.829,Z 842.353,A -85,B 0,C 180,E1 -29642.448,E2 -29642.448} C_VEL
LIN {X 0,Y 147.014,Z 839.24,A -85,B 0,C 180,E1 -29639.955,E2 -29639.955} C_VEL
LIN {X 0,Y 143.827,Z 837.094,A -85,B 0,C 180,E1 -29638.157,E2 -29638.157} C_VEL
LIN {X 0,Y 143.035,Z 836.417,A -85,B 0,C 180,E1 -29637.481,E2 -29637.481} C_VEL
LIN {X 0,Y 139.685,Z 832.529,A -85,B 0,C 180,E1 -29633.651,E2 -29633.651} C_VEL
LIN {X 0,Y 137.308,Z 827.692,A -85,B 0,C 180,E1 -29629.366,E2 -29629.366} C_VEL
LIN {X 0,Y 135.815,Z 820.958,A -85,B 0,C 180,E1 -29624.181,E2 -29624.181} C_VEL
LIN {X 0,Y 135.789,Z 814.729,A -85,B 0,C 180,E1 -29620.016,E2 -29620.016} C_VEL
LIN {X 0,Y 136.224,Z 808.279,A -85,B 0,C 180,E1 -29616.385,E2 -29616.385} C_VEL
LIN {X 0,Y 136.292,Z 802.232,A -85,B 0,C 180,E1 -29613.684,E2 -29613.684} C_VEL
LIN {X 0,Y 135.932,Z 792.093,A -85,B 0,C 180,E1 -29610.001,E2 -29610.001} C_VEL
LIN {X 0,Y 135.814,Z 780.516,A -85,B 0,C 180,E1 -29606.674,E2 -29606.674} C_VEL
LIN {X 0,Y 135.964,Z 769.153,A -85,B 0,C 180,E1 -29604.087,E2 -29604.087} C_VEL
LIN {X 0,Y 136.072,Z 758.985,A -85,B 0,C 180,E1 -29602.235,E2 -29602.235} C_VEL
LIN {X 0,Y 136.177,Z 747.658,A -85,B 0,C 180,E1 -29600.629,E2 -29600.629} C_VEL
LIN {X 0,Y 136.458,Z 721.537,A -85,B 0,C 180,E1 -29597.873,E2 -29597.873} C_VEL
LIN {X 0,Y 136.546,Z 689.327,A -85,B 0,C 180,E1 -29594.711,E2 -29594.711} C_VEL
LIN {X 0,Y 133.798,Z 656.711,A -85,B 0,C 180,E1 -29591.793,E2 -29591.793} C_VEL
LIN {X 0,Y 133.393,Z 640.798,A -85,B 0,C 180,E1 -29590.254,E2 -29590.254} C_VEL
LIN {X 0,Y 133.652,Z 640.772,A -85,B 0,C 180,E1 -29585.212,E2 -29585.212} C_VEL
LIN {X 0,Y 133.466,Z 640.784,A -85,B 0,C 180,E1 -29581.815,E2 -29581.815} C_VEL
LIN {X 0,Y 133.212,Z 640.823,A -85,B 0,C 180,E1 -29577.278,E2 -29577.278} C_VEL
LIN {X 0,Y 133.106,Z 640.827,A -85,B 0,C 180,E1 -29570.842,E2 -29570.842} C_VEL
LIN {X 0,Y 133.138,Z 640.832,A -85,B 0,C 180,E1 -29566.849,E2 -29566.849} C_VEL
LIN {X 0,Y 133.144,Z 640.826,A -85,B 0,C 180,E1 -29562.566,E2 -29562.566} C_VEL
LIN {X 0,Y 133.109,Z 640.837,A -85,B 0,C 180,E1 -29557.878,E2 -29557.878} C_VEL
LIN {X 0,Y 133.186,Z 640.818,A -85,B 0,C 180,E1 -29551.731,E2 -29551.731} C_VEL
LIN {X 0,Y 133.23,Z 640.821,A -85,B 0,C 180,E1 -29546.651,E2 -29546.651} C_VEL
LIN {X 0,Y 133.312,Z 640.809,A -85,B 0,C 180,E1 -29538.96,E2 -29538.96} C_VEL
LIN {X 0,Y 133.482,Z 640.781,A -85,B 0,C 180,E1 -29532.117,E2 -29532.117} C_VEL
LIN {X 0,Y 133.995,Z 640.726,A -85,B 0,C 180,E1 -29526.002,E2 -29526.002} C_VEL
LIN {X 0,Y 134.315,Z 640.683,A -85,B 0,C 180,E1 -29520.001,E2 -29520.001} C_VEL
LIN {X 0,Y 133.981,Z 640.719,A -85,B 0,C 180,E1 -29513.364,E2 -29513.364} C_VEL
LIN {X 0,Y 133.492,Z 640.79,A -85,B 0,C 180,E1 -29507.886,E2 -29507.886} C_VEL
LIN {X 0,Y 133.335,Z 640.804,A -85,B 0,C 180,E1 -29501.01,E2 -29501.01} C_VEL
LIN {X 0,Y 133.235,Z 640.811,A -85,B 0,C 180,E1 -29493.344,E2 -29493.344} C_VEL
LIN {X 0,Y 133.192,Z 640.825,A -85,B 0,C 180,E1 -29487.29,E2 -29487.29} C_VEL
LIN {X 0,Y 133.128,Z 640.831,A -85,B 0,C 180,E1 -29480.85,E2 -29480.85} C_VEL
LIN {X 0,Y 133.176,Z 640.827,A -85,B 0,C 180,E1 -29476.865,E2 -29476.865} C_VEL
LIN {X 0,Y 133.173,Z 640.821,A -85,B 0,C 180,E1 -29472.58,E2 -29472.58} C_VEL
LIN {X 0,Y 133.163,Z 640.83,A -85,B 0,C 180,E1 -29467.909,E2 -29467.909} C_VEL
LIN {X 0,Y 133.238,Z 640.818,A -85,B 0,C 180,E1 -29461.715,E2 -29461.715} C_VEL
LIN {X 0,Y 133.226,Z 640.814,A -85,B 0,C 180,E1 -29454.872,E2 -29454.872} C_VEL
LIN {X 0,Y 133.422,Z 640.798,A -85,B 0,C 180,E1 -29448.36,E2 -29448.36} C_VEL
LIN {X 0,Y 133.515,Z 640.783,A -85,B 0,C 180,E1 -29442.113,E2 -29442.113} C_VEL
LIN {X 0,Y 133.992,Z 640.719,A -85,B 0,C 180,E1 -29436.001,E2 -29436.001} C_VEL
LIN {X 0,Y 134.314,Z 640.688,A -85,B 0,C 180,E1 -29429.999,E2 -29429.999} C_VEL
LIN {X 0,Y 133.98,Z 640.725,A -85,B 0,C 180,E1 -29423.362,E2 -29423.362} C_VEL
LIN {X 0,Y 133.515,Z 640.783,A -85,B 0,C 180,E1 -29417.886,E2 -29417.886} C_VEL
LIN {X 0,Y 133.423,Z 640.798,A -85,B 0,C 180,E1 -29411.639,E2 -29411.639} C_VEL
LIN {X 0,Y 133.226,Z 640.814,A -85,B 0,C 180,E1 -29405.127,E2 -29405.127} C_VEL
LIN {X 0,Y 133.146,Z 640.833,A -85,B 0,C 180,E1 -29401.74,E2 -29401.74} C_VEL
LIN {X 0,Y 133.153,Z 640.825,A -85,B 0,C 180,E1 -29397.314,E2 -29397.314} C_VEL
LIN {X 0,Y 133.114,Z 640.836,A -85,B 0,C 180,E1 -29390.843,E2 -29390.843} C_VEL
LIN {X 0,Y 133.177,Z 640.82,A -85,B 0,C 180,E1 -29386.863,E2 -29386.863} C_VEL
LIN {X 0,Y 133.175,Z 640.827,A -85,B 0,C 180,E1 -29382.578,E2 -29382.578} C_VEL
LIN {X 0,Y 133.416,Z 640.793,A -85,B 0,C 180,E1 -29375.274,E2 -29375.274} C_VEL
LIN {X 0,Y 134.215,Z 640.702,A -85,B 0,C 180,E1 -29369.173,E2 -29369.173} C_VEL
LIN {X 0,Y 136.79,Z 670.429,A -85,B 0,C 180,E1 -29366.515,E2 -29366.515} C_VEL
LIN {X 0,Y 135.759,Z 734.34,A -85,B 0,C 180,E1 -29360.164,E2 -29360.164} C_VEL
LIN {X 0,Y 135.509,Z 748.332,A -85,B 0,C 180,E1 -29358.436,E2 -29358.436} C_VEL
LIN {X 0,Y 135.083,Z 760.411,A -85,B 0,C 180,E1 -29356.376,E2 -29356.376} C_VEL
LIN {X 0,Y 134.894,Z 770.268,A -85,B 0,C 180,E1 -29354.278,E2 -29354.278} C_VEL
LIN {X 0,Y 134.758,Z 779.112,A -85,B 0,C 180,E1 -29351.999,E2 -29351.999} C_VEL
LIN {X 0,Y 134.668,Z 789.36,A -85,B 0,C 180,E1 -29348.79,E2 -29348.79} C_VEL
LIN {X 0,Y 134.522,Z 796.85,A -85,B 0,C 180,E1 -29345.977,E2 -29345.977} C_VEL
LIN {X 0,Y 134.383,Z 805.488,A -85,B 0,C 180,E1 -29342.046,E2 -29342.046} C_VEL
LIN {X 0,Y 134.82,Z 813.341,A -85,B 0,C 180,E1 -29337.766,E2 -29337.766} C_VEL
LIN {X 0,Y 136.49,Z 821.29,A -85,B 0,C 180,E1 -29332.628,E2 -29332.628} C_VEL
LIN {X 0,Y 138.879,Z 827.086,A -85,B 0,C 180,E1 -29328.36,E2 -29328.36} C_VEL
LIN {X 0,Y 142.294,Z 832.017,A -85,B 0,C 180,E1 -29324.291,E2 -29324.291} C_VEL
LIN {X 0,Y 148.424,Z 837.288,A -85,B 0,C 180,E1 -29319.271,E2 -29319.271} C_VEL
LIN {X 0,Y 153.855,Z 840.437,A -85,B 0,C 180,E1 -29315.811,E2 -29315.811} C_VEL
LIN {X 0,Y 162.476,Z 843.38,A -85,B 0,C 180,E1 -29311.691,E2 -29311.691} C_VEL
LIN {X 0,Y 172.239,Z 845.035,A -85,B 0,C 180,E1 -29308.084,E2 -29308.084} C_VEL
LIN {X 0,Y 177.449,Z 845.454,A -85,B 0,C 180,E1 -29306.452,E2 -29306.452} C_VEL
LIN {X 0,Y 188.549,Z 845.082,A -85,B 0,C 180,E1 -29303.531,E2 -29303.531} C_VEL
LIN {X 0,Y 201.093,Z 843.027,A -85,B 0,C 180,E1 -29300.854,E2 -29300.854} C_VEL
LIN {X 0,Y 200.209,Z 843.298,A -85,B 0,C 180,E1 -29300.326,E2 -29300.326} C_VEL
LIN {X 0,Y 188.743,Z 845.559,A -85,B 0,C 180,E1 -29297.922,E2 -29297.922} C_VEL
LIN {X 0,Y 177.945,Z 846.486,A -85,B 0,C 180,E1 -29295.116,E2 -29295.116} C_VEL
LIN {X 0,Y 167.91,Z 846.144,A -85,B 0,C 180,E1 -29291.871,E2 -29291.871} C_VEL
LIN {X 0,Y 157.406,Z 844.131,A -85,B 0,C 180,E1 -29287.421,E2 -29287.421} C_VEL
LIN {X 0,Y 151.032,Z 841.807,A -85,B 0,C 180,E1 -29283.817,E2 -29283.817} C_VEL
LIN {X 0,Y 144.594,Z 837.807,A -85,B 0,C 180,E1 -29278.975,E2 -29278.975} C_VEL
LIN {X 0,Y 143.035,Z 836.417,A -85,B 0,C 180,E1 -29277.481,E2 -29277.481} C_VEL
LIN {X 0,Y 140.542,Z 834.291,A -85,B 0,C 180,E1 -29275.512,E2 -29275.512} C_VEL
LIN {X 0,Y 135.588,Z 829.632,A -85,B 0,C 180,E1 -29272.511,E2 -29272.511} C_VEL
LIN {X 0,Y 131.356,Z 824.349,A -85,B 0,C 180,E1 -29269.386,E2 -29269.386} C_VEL
LIN {X 0,Y 130.079,Z 821.159,A -85,B 0,C 180,E1 -29267.265,E2 -29267.265} C_VEL
LIN {X 0,Y 129.481,Z 814.477,A -85,B 0,C 180,E1 -29262.497,E2 -29262.497} C_VEL
LIN {X 0,Y 129.81,Z 808.105,A -85,B 0,C 180,E1 -29258.534,E2 -29258.534} C_VEL
LIN {X 0,Y 130.025,Z 801.713,A -85,B 0,C 180,E1 -29255.41,E2 -29255.41} C_VEL
LIN {X 0,Y 129.587,Z 791.624,A -85,B 0,C 180,E1 -29251.549,E2 -29251.549} C_VEL
LIN {X 0,Y 129.37,Z 780.124,A -85,B 0,C 180,E1 -29248.061,E2 -29248.061} C_VEL
LIN {X 0,Y 129.382,Z 768.992,A -85,B 0,C 180,E1 -29245.343,E2 -29245.343} C_VEL
LIN {X 0,Y 129.426,Z 759.102,A -85,B 0,C 180,E1 -29243.397,E2 -29243.397} C_VEL
LIN {X 0,Y 129.473,Z 748.305,A -85,B 0,C 180,E1 -29241.738,E2 -29241.738} C_VEL
LIN {X 0,Y 129.633,Z 723.723,A -85,B 0,C 180,E1 -29238.978,E2 -29238.978} C_VEL
LIN {X 0,Y 129.644,Z 689.621,A -85,B 0,C 180,E1 -29235.431,E2 -29235.431} C_VEL
LIN {X 0,Y 126.844,Z 657.559,A -85,B 0,C 180,E1 -29232.423,E2 -29232.423} C_VEL
LIN {X 0,Y 126.38,Z 641.672,A -85,B 0,C 180,E1 -29230.799,E2 -29230.799} C_VEL
LIN {X 0,Y 126.584,Z 641.647,A -85,B 0,C 180,E1 -29223.726,E2 -29223.726} C_VEL
LIN {X 0,Y 126.108,Z 641.709,A -85,B 0,C 180,E1 -29216.26,E2 -29216.26} C_VEL
LIN {X 0,Y 126.074,Z 641.702,A -85,B 0,C 180,E1 -29211.062,E2 -29211.062} C_VEL
LIN {X 0,Y 126.066,Z 641.715,A -85,B 0,C 180,E1 -29206.246,E2 -29206.246} C_VEL
LIN {X 0,Y 126.05,Z 641.707,A -85,B 0,C 180,E1 -29201.824,E2 -29201.824} C_VEL
LIN {X 0,Y 126.056,Z 641.716,A -85,B 0,C 180,E1 -29197.679,E2 -29197.679} C_VEL
LIN {X 0,Y 126.088,Z 641.706,A -85,B 0,C 180,E1 -29193.564,E2 -29193.564} C_VEL
LIN {X 0,Y 126.145,Z 641.704,A -85,B 0,C 180,E1 -29187.324,E2 -29187.324} C_VEL
LIN {X 0,Y 126.111,Z 641.702,A -85,B 0,C 180,E1 -29182.88,E2 -29182.88} C_VEL
LIN {X 0,Y 126.24,Z 641.691,A -85,B 0,C 180,E1 -29179.397,E2 -29179.397} C_VEL
LIN {X 0,Y 126.384,Z 641.666,A -85,B 0,C 180,E1 -29172.809,E2 -29172.809} C_VEL
LIN {X 0,Y 126.943,Z 641.605,A -85,B 0,C 180,E1 -29166.337,E2 -29166.337} C_VEL
LIN {X 0,Y 127.284,Z 641.559,A -85,B 0,C 180,E1 -29160.001,E2 -29160.001} C_VEL
LIN {X 0,Y 126.923,Z 641.598,A -85,B 0,C 180,E1 -29153.387,E2 -29153.387} C_VEL
LIN {X 0,Y 126.397,Z 641.672,A -85,B 0,C 180,E1 -29147.194,E2 -29147.194} C_VEL
LIN {X 0,Y 126.272,Z 641.685,A -85,B 0,C 180,E1 -29140.561,E2 -29140.561} C_VEL
LIN {X 0,Y 126.182,Z 641.69,A -85,B 0,C 180,E1 -29133.636,E2 -29133.636} C_VEL
LIN {X 0,Y 126.094,Z 641.709,A -85,B 0,C 180,E1 -29130.005,E2 -29130.005} C_VEL
LIN {X 0,Y 126.092,Z 641.709,A -85,B 0,C 180,E1 -29126.256,E2 -29126.256} C_VEL
LIN {X 0,Y 126.097,Z 641.707,A -85,B 0,C 180,E1 -29121.047,E2 -29121.047} C_VEL
LIN {X 0,Y 126.098,Z 641.707,A -85,B 0,C 180,E1 -29116.229,E2 -29116.229} C_VEL
LIN {X 0,Y 126.079,Z 641.708,A -85,B 0,C 180,E1 -29111.81,E2 -29111.81} C_VEL
LIN {X 0,Y 126.106,Z 641.708,A -85,B 0,C 180,E1 -29107.66,E2 -29107.66} C_VEL
LIN {X 0,Y 126.143,Z 641.696,A -85,B 0,C 180,E1 -29103.603,E2 -29103.603} C_VEL
LIN {X 0,Y 126.172,Z 641.699,A -85,B 0,C 180,E1 -29097.35,E2 -29097.35} C_VEL
LIN {X 0,Y 126.162,Z 641.696,A -85,B 0,C 180,E1 -29092.869,E2 -29092.869} C_VEL
LIN {X 0,Y 126.309,Z 641.684,A -85,B 0,C 180,E1 -29089.434,E2 -29089.434} C_VEL
LIN {X 0,Y 126.42,Z 641.665,A -85,B 0,C 180,E1 -29082.804,E2 -29082.804} C_VEL
LIN {X 0,Y 126.94,Z 641.599,A -85,B 0,C 180,E1 -29076.335,E2 -29076.335} C_VEL
LIN {X 0,Y 127.283,Z 641.564,A -85,B 0,C 180,E1 -29069.999,E2 -29069.999} C_VEL
LIN {X 0,Y 126.922,Z 641.603,A -85,B 0,C 180,E1 -29063.386,E2 -29063.386} C_VEL
LIN {X 0,Y 126.421,Z 641.665,A -85,B 0,C 180,E1 -29057.195,E2 -29057.195} C_VEL
LIN {X 0,Y 126.299,Z 641.685,A -85,B 0,C 180,E1 -29050.525,E2 -29050.525} C_VEL
LIN {X 0,Y 126.185,Z 641.695,A -85,B 0,C 180,E1 -29043.635,E2 -29043.635} C_VEL
LIN {X 0,Y 126.087,Z 641.703,A -85,B 0,C 180,E1 -29036.436,E2 -29036.436} C_VEL
LIN {X 0,Y 126.08,Z 641.712,A -85,B 0,C 180,E1 -29031.055,E2 -29031.055} C_VEL
LIN {X 0,Y 126.1,Z 641.701,A -85,B 0,C 180,E1 -29026.227,E2 -29026.227} C_VEL
LIN {X 0,Y 126.092,Z 641.712,A -85,B 0,C 180,E1 -29021.804,E2 -29021.804} C_VEL
LIN {X 0,Y 126.199,Z 641.69,A -85,B 0,C 180,E1 -29017.627,E2 -29017.627} C_VEL
LIN {X 0,Y 126.561,Z 641.652,A -85,B 0,C 180,E1 -29013.602,E2 -29013.602} C_VEL
LIN {X 0,Y 127.249,Z 641.567,A -85,B 0,C 180,E1 -29008.68,E2 -29008.68} C_VEL
LIN {X 0,Y 129.731,Z 668.181,A -85,B 0,C 180,E1 -29006.152,E2 -29006.152} C_VEL
LIN {X 0,Y 129.169,Z 713.579,A -85,B 0,C 180,E1 -29001.438,E2 -29001.438} C_VEL
LIN {X 0,Y 128.948,Z 740.858,A -85,B 0,C 180,E1 -28998.404,E2 -28998.404} C_VEL
LIN {X 0,Y 128.723,Z 751.574,A -85,B 0,C 180,E1 -28996.802,E2 -28996.802} C_VEL
LIN {X 0,Y 128.439,Z 762.925,A -85,B 0,C 180,E1 -28994.608,E2 -28994.608} C_VEL
LIN {X 0,Y 128.337,Z 773.138,A -85,B 0,C 180,E1 -28992.169,E2 -28992.169} C_VEL
LIN {X 0,Y 128.228,Z 782.515,A -85,B 0,C 180,E1 -28989.431,E2 -28989.431} C_VEL
LIN {X 0,Y 128.184,Z 789.434,A -85,B 0,C 180,E1 -28987.062,E2 -28987.062} C_VEL
LIN {X 0,Y 128.093,Z 797.951,A -85,B 0,C 180,E1 -28983.598,E2 -28983.598} C_VEL
LIN {X 0,Y 128.21,Z 806.632,A -85,B 0,C 180,E1 -28979.216,E2 -28979.216} C_VEL
LIN {X 0,Y 129.136,Z 814.495,A -85,B 0,C 180,E1 -28974.552,E2 -28974.552} C_VEL
LIN {X 0,Y 131.021,Z 821.262,A -85,B 0,C 180,E1 -28969.993,E2 -28969.993} C_VEL
LIN {X 0,Y 134.454,Z 827.812,A -85,B 0,C 180,E1 -28964.901,E2 -28964.901} C_VEL
LIN {X 0,Y 138.571,Z 832.633,A -85,B 0,C 180,E1 -28960.818,E2 -28960.818} C_VEL
LIN {X 0,Y 143.651,Z 836.741,A -85,B 0,C 180,E1 -28957.04,E2 -28957.04} C_VEL
LIN {X 0,Y 151.668,Z 840.859,A -85,B 0,C 180,E1 -28952.494,E2 -28952.494} C_VEL
LIN {X 0,Y 161.004,Z 843.742,A -85,B 0,C 180,E1 -28948.529,E2 -28948.529} C_VEL
LIN {X 0,Y 169.906,Z 845.208,A -85,B 0,C 180,E1 -28945.54,E2 -28945.54} C_VEL
LIN {X 0,Y 176.936,Z 845.723,A -85,B 0,C 180,E1 -28943.571,E2 -28943.571} C_VEL
LIN {X 0,Y 188.647,Z 845.251,A -85,B 0,C 180,E1 -28940.86,E2 -28940.86} C_VEL
LIN {X 0,Y 184.053,Z 845.746,A -85,B 0,C 180,E1 -28939.565,E2 -28939.565} C_VEL
LIN {X 0,Y 178.424,Z 846.157,A -85,B 0,C 180,E1 -28938.236,E2 -28938.236} C_VEL
LIN {X 0,Y 167.788,Z 845.99,A -85,B 0,C 180,E1 -28935.209,E2 -28935.209} C_VEL
LIN {X 0,Y 157.894,Z 844.596,A -85,B 0,C 180,E1 -28931.716,E2 -28931.716} C_VEL
LIN {X 0,Y 149.251,Z 842.043,A -85,B 0,C 180,E1 -28927.597,E2 -28927.597} C_VEL
LIN {X 0,Y 141.848,Z 838.28,A -85,B 0,C 180,E1 -28922.901,E2 -28922.901} C_VEL
LIN {X 0,Y 135.925,Z 833.197,A -85,B 0,C 180,E1 -28917.632,E2 -28917.632} C_VEL
LIN {X 0,Y 132.617,Z 828.659,A -85,B 0,C 180,E1 -28913.337,E2 -28913.337} C_VEL
LIN {X 0,Y 130.079,Z 821.159,A -85,B 0,C 180,E1 -28907.265,E2 -28907.265} C_VEL
LIN {X 0,Y 129.14,Z 817.982,A -85,B 0,C 180,E1 -28905.146,E2 -28905.146} C_VEL
LIN {X 0,Y 127.687,Z 814.245,A -85,B 0,C 180,E1 -28903.192,E2 -28903.192} C_VEL
LIN {X 0,Y 124.658,Z 805.931,A -85,B 0,C 180,E1 -28899.471,E2 -28899.471} C_VEL
LIN {X 0,Y 123.78,Z 800.226,A -85,B 0,C 180,E1 -28896.9,E2 -28896.9} C_VEL
LIN {X 0,Y 123.369,Z 791.165,A -85,B 0,C 180,E1 -28893.255,E2 -28893.255} C_VEL
LIN {X 0,Y 123.019,Z 779.675,A -85,B 0,C 180,E1 -28889.593,E2 -28889.593} C_VEL
LIN {X 0,Y 122.934,Z 768.565,A -85,B 0,C 180,E1 -28886.734,E2 -28886.734} C_VEL
LIN {X 0,Y 122.904,Z 758.672,A -85,B 0,C 180,E1 -28884.687,E2 -28884.687} C_VEL
LIN {X 0,Y 122.892,Z 747.954,A -85,B 0,C 180,E1 -28882.941,E2 -28882.941} C_VEL
LIN {X 0,Y 122.902,Z 723.228,A -85,B 0,C 180,E1 -28879.959,E2 -28879.959} C_VEL
LIN {X 0,Y 122.759,Z 689.625,A -85,B 0,C 180,E1 -28876.207,E2 -28876.207} C_VEL
LIN {X 0,Y 119.867,Z 657.198,A -85,B 0,C 180,E1 -28873.012,E2 -28873.012} C_VEL
LIN {X 0,Y 119.408,Z 642.542,A -85,B 0,C 180,E1 -28871.399,E2 -28871.399} C_VEL
LIN {X 0,Y 119.402,Z 642.547,A -85,B 0,C 180,E1 -28865.756,E2 -28865.756} C_VEL
LIN {X 0,Y 119.353,Z 642.541,A -85,B 0,C 180,E1 -28861.68,E2 -28861.68} C_VEL
LIN {X 0,Y 118.983,Z 642.594,A -85,B 0,C 180,E1 -28853.936,E2 -28853.936} C_VEL
LIN {X 0,Y 118.989,Z 642.589,A -85,B 0,C 180,E1 -28849.645,E2 -28849.645} C_VEL
LIN {X 0,Y 118.995,Z 642.594,A -85,B 0,C 180,E1 -28844.941,E2 -28844.941} C_VEL
LIN {X 0,Y 118.992,Z 642.587,A -85,B 0,C 180,E1 -28840.073,E2 -28840.073} C_VEL
LIN {X 0,Y 119.004,Z 642.593,A -85,B 0,C 180,E1 -28834.511,E2 -28834.511} C_VEL
LIN {X 0,Y 119.075,Z 642.584,A -85,B 0,C 180,E1 -28828.074,E2 -28828.074} C_VEL
LIN {X 0,Y 119.046,Z 642.586,A -85,B 0,C 180,E1 -28824.323,E2 -28824.323} C_VEL
LIN {X 0,Y 119.147,Z 642.571,A -85,B 0,C 180,E1 -28819.846,E2 -28819.846} C_VEL
LIN {X 0,Y 119.29,Z 642.551,A -85,B 0,C 180,E1 -28813.585,E2 -28813.585} C_VEL
LIN {X 0,Y 119.863,Z 642.487,A -85,B 0,C 180,E1 -28806.576,E2 -28806.576} C_VEL
LIN {X 0,Y 120.251,Z 642.435,A -85,B 0,C 180,E1 -28800.001,E2 -28800.001} C_VEL
LIN {X 0,Y 119.849,Z 642.479,A -85,B 0,C 180,E1 -28793.289,E2 -28793.289} C_VEL
LIN {X 0,Y 119.304,Z 642.556,A -85,B 0,C 180,E1 -28786.419,E2 -28786.419} C_VEL
LIN {X 0,Y 119.177,Z 642.57,A -85,B 0,C 180,E1 -28780.113,E2 -28780.113} C_VEL
LIN {X 0,Y 119.056,Z 642.584,A -85,B 0,C 180,E1 -28775.681,E2 -28775.681} C_VEL
LIN {X 0,Y 119.073,Z 642.578,A -85,B 0,C 180,E1 -28771.928,E2 -28771.928} C_VEL
LIN {X 0,Y 119.012,Z 642.588,A -85,B 0,C 180,E1 -28765.483,E2 -28765.483} C_VEL
LIN {X 0,Y 119.031,Z 642.591,A -85,B 0,C 180,E1 -28759.663,E2 -28759.663} C_VEL
LIN {X 0,Y 119.048,Z 642.582,A -85,B 0,C 180,E1 -28754.913,E2 -28754.913} C_VEL
LIN {X 0,Y 119.039,Z 642.589,A -85,B 0,C 180,E1 -28750.101,E2 -28750.101} C_VEL
LIN {X 0,Y 119.045,Z 642.58,A -85,B 0,C 180,E1 -28744.542,E2 -28744.542} C_VEL
LIN {X 0,Y 119.107,Z 642.581,A -85,B 0,C 180,E1 -28738.064,E2 -28738.064} C_VEL
LIN {X 0,Y 119.166,Z 642.572,A -85,B 0,C 180,E1 -28730.65,E2 -28730.65} C_VEL
LIN {X 0,Y 119.242,Z 642.561,A -85,B 0,C 180,E1 -28727.079,E2 -28727.079} C_VEL
LIN {X 0,Y 119.505,Z 642.532,A -85,B 0,C 180,E1 -28720.127,E2 -28720.127} C_VEL
LIN {X 0,Y 119.874,Z 642.481,A -85,B 0,C 180,E1 -28716.631,E2 -28716.631} C_VEL
LIN {X 0,Y 120.251,Z 642.44,A -85,B 0,C 180,E1 -28709.999,E2 -28709.999} C_VEL
LIN {X 0,Y 119.848,Z 642.485,A -85,B 0,C 180,E1 -28703.287,E2 -28703.287} C_VEL
LIN {X 0,Y 119.329,Z 642.546,A -85,B 0,C 180,E1 -28696.42,E2 -28696.42} C_VEL
LIN {X 0,Y 119.216,Z 642.568,A -85,B 0,C 180,E1 -28690.059,E2 -28690.059} C_VEL
LIN {X 0,Y 119.075,Z 642.575,A -85,B 0,C 180,E1 -28685.683,E2 -28685.683} C_VEL
LIN {X 0,Y 119.074,Z 642.585,A -85,B 0,C 180,E1 -28681.926,E2 -28681.926} C_VEL
LIN {X 0,Y 119.003,Z 642.585,A -85,B 0,C 180,E1 -28675.488,E2 -28675.488} C_VEL
LIN {X 0,Y 118.995,Z 642.593,A -85,B 0,C 180,E1 -28669.646,E2 -28669.646} C_VEL
LIN {X 0,Y 119.049,Z 642.582,A -85,B 0,C 180,E1 -28664.912,E2 -28664.912} C_VEL
LIN {X 0,Y 119.058,Z 642.587,A -85,B 0,C 180,E1 -28660.108,E2 -28660.108} C_VEL
LIN {X 0,Y 119.681,Z 642.511,A -85,B 0,C 180,E1 -28651.784,E2 -28651.784} C_VEL
LIN {X 0,Y 120.292,Z 642.432,A -85,B 0,C 180,E1 -28648.042,E2 -28648.042} C_VEL
LIN {X 0,Y 122.836,Z 670.513,A -85,B 0,C 180,E1 -28645.262,E2 -28645.262} C_VEL
LIN {X 0,Y 122.382,Z 731.766,A -85,B 0,C 180,E1 -28638.347,E2 -28638.347} C_VEL
LIN {X 0,Y 122.201,Z 747.549,A -85,B 0,C 180,E1 -28636.225,E2 -28636.225} C_VEL
LIN {X 0,Y 121.932,Z 760.59,A -85,B 0,C 180,E1 -28633.706,E2 -28633.706} C_VEL
LIN {X 0,Y 121.868,Z 771.054,A -85,B 0,C 180,E1 -28631.173,E2 -28631.173} C_VEL
LIN {X 0,Y 121.842,Z 779.676,A -85,B 0,C 180,E1 -28628.652,E2 -28628.652} C_VEL
LIN {X 0,Y 121.823,Z 787.934,A -85,B 0,C 180,E1 -28625.774,E2 -28625.774} C_VEL
LIN {X 0,Y 121.867,Z 797.398,A -85,B 0,C 180,E1 -28621.646,E2 -28621.646} C_VEL
LIN {X 0,Y 122.236,Z 806.603,A -85,B 0,C 180,E1 -28616.714,E2 -28616.714} C_VEL
LIN {X 0,Y 123.53,Z 814.448,A -85,B 0,C 180,E1 -28611.85,E2 -28611.85} C_VEL
LIN {X 0,Y 125.86,Z 821.064,A -85,B 0,C 180,E1 -28607.137,E2 -28607.137} C_VEL
LIN {X 0,Y 130.618,Z 828.496,A -85,B 0,C 180,E1 -28601.23,E2 -28601.23} C_VEL
LIN {X 0,Y 135.482,Z 833.246,A -85,B 0,C 180,E1 -28597.184,E2 -28597.184} C_VEL
LIN {X 0,Y 141.122,Z 837.179,A -85,B 0,C 180,E1 -28593.467,E2 -28593.467} C_VEL
LIN {X 0,Y 149.981,Z 841.266,A -85,B 0,C 180,E1 -28589.087,E2 -28589.087} C_VEL
LIN {X 0,Y 154.89,Z 842.86,A -85,B 0,C 180,E1 -28587.134,E2 -28587.134} C_VEL
LIN {X 0,Y 165.455,Z 845.08,A -85,B 0,C 180,E1 -28583.652,E2 -28583.652} C_VEL
LIN {X 0,Y 176.013,Z 845.956,A -85,B 0,C 180,E1 -28580.919,E2 -28580.919} C_VEL
LIN {X 0,Y 175.105,Z 845.975,A -85,B 0,C 180,E1 -28580.304,E2 -28580.304} C_VEL
LIN {X 0,Y 162.888,Z 845.262,A -85,B 0,C 180,E1 -28576.973,E2 -28576.973} C_VEL
LIN {X 0,Y 157.693,Z 844.534,A -85,B 0,C 180,E1 -28575.292,E2 -28575.292} C_VEL
LIN {X 0,Y 148.06,Z 842.126,A -85,B 0,C 180,E1 -28571.477,E2 -28571.477} C_VEL
LIN {X 0,Y 139.773,Z 838.573,A -85,B 0,C 180,E1 -28566.968,E2 -28566.968} C_VEL
LIN {X 0,Y 132.853,Z 833.803,A -85,B 0,C 180,E1 -28561.819,E2 -28561.819} C_VEL
LIN {X 0,Y 127.611,Z 827.633,A -85,B 0,C 180,E1 -28556.048,E2 -28556.048} C_VEL
LIN {X 0,Y 124.71,Z 821.253,A -85,B 0,C 180,E1 -28550.551,E2 -28550.551} C_VEL
LIN {X 0,Y 123.468,Z 814.225,A -85,B 0,C 180,E1 -28545.327,E2 -28545.327} C_VEL
LIN {X 0,Y 123.675,Z 805.678,A -85,B 0,C 180,E1 -28539.783,E2 -28539.783} C_VEL
LIN {X 0,Y 123.78,Z 800.226,A -85,B 0,C 180,E1 -28536.9,E2 -28536.9} C_VEL
LIN {X 0,Y 123.475,Z 797.327,A -85,B 0,C 180,E1 -28535.702,E2 -28535.702} C_VEL
LIN {X 0,Y 122.697,Z 794.199,A -85,B 0,C 180,E1 -28534.671,E2 -28534.671} C_VEL
LIN {X 0,Y 120.352,Z 787.575,A -85,B 0,C 180,E1 -28532.962,E2 -28532.962} C_VEL
LIN {X 0,Y 117.382,Z 778.908,A -85,B 0,C 180,E1 -28530.984,E2 -28530.984} C_VEL
LIN {X 0,Y 116.587,Z 773.409,A -85,B 0,C 180,E1 -28529.619,E2 -28529.619} C_VEL
LIN {X 0,Y 116.473,Z 760.528,A -85,B 0,C 180,E1 -28526.553,E2 -28526.553} C_VEL
LIN {X 0,Y 116.367,Z 748.235,A -85,B 0,C 180,E1 -28524.387,E2 -28524.387} C_VEL
LIN {X 0,Y 116.256,Z 725.462,A -85,B 0,C 180,E1 -28521.447,E2 -28521.447} C_VEL
LIN {X 0,Y 115.967,Z 689.568,A -85,B 0,C 180,E1 -28517.187,E2 -28517.187} C_VEL
LIN {X 0,Y 112.956,Z 657.19,A -85,B 0,C 180,E1 -28513.797,E2 -28513.797} C_VEL
LIN {X 0,Y 112.481,Z 643.404,A -85,B 0,C 180,E1 -28512.211,E2 -28512.211} C_VEL
LIN {X 0,Y 112.303,Z 643.427,A -85,B 0,C 180,E1 -28504.114,E2 -28504.114} C_VEL
LIN {X 0,Y 112.141,Z 643.439,A -85,B 0,C 180,E1 -28500.021,E2 -28500.021} C_VEL
LIN {X 0,Y 111.967,Z 643.47,A -85,B 0,C 180,E1 -28494.417,E2 -28494.417} C_VEL
LIN {X 0,Y 111.882,Z 643.477,A -85,B 0,C 180,E1 -28488.701,E2 -28488.701} C_VEL
LIN {X 0,Y 111.891,Z 643.475,A -85,B 0,C 180,E1 -28483.521,E2 -28483.521} C_VEL
LIN {X 0,Y 111.894,Z 643.476,A -85,B 0,C 180,E1 -28478.756,E2 -28478.756} C_VEL
LIN {X 0,Y 111.946,Z 643.47,A -85,B 0,C 180,E1 -28474.274,E2 -28474.274} C_VEL
LIN {X 0,Y 111.968,Z 643.467,A -85,B 0,C 180,E1 -28468.861,E2 -28468.861} C_VEL
LIN {X 0,Y 112.002,Z 643.456,A -85,B 0,C 180,E1 -28462.04,E2 -28462.04} C_VEL
LIN {X 0,Y 112.102,Z 643.453,A -85,B 0,C 180,E1 -28458.206,E2 -28458.206} C_VEL
LIN {X 0,Y 112.363,Z 643.414,A -85,B 0,C 180,E1 -28450.78,E2 -28450.78} C_VEL
LIN {X 0,Y 112.821,Z 643.364,A -85,B 0,C 180,E1 -28446.616,E2 -28446.616} C_VEL
LIN {X 0,Y 113.217,Z 643.311,A -85,B 0,C 180,E1 -28440.001,E2 -28440.001} C_VEL
LIN {X 0,Y 112.714,Z 643.367,A -85,B 0,C 180,E1 -28432.862,E2 -28432.862} C_VEL
LIN {X 0,Y 112.2,Z 643.438,A -85,B 0,C 180,E1 -28425.541,E2 -28425.541} C_VEL
LIN {X 0,Y 112.118,Z 643.452,A -85,B 0,C 180,E1 -28419.57,E2 -28419.57} C_VEL
LIN {X 0,Y 111.956,Z 643.462,A -85,B 0,C 180,E1 -28414.028,E2 -28414.028} C_VEL
LIN {X 0,Y 111.936,Z 643.473,A -85,B 0,C 180,E1 -28409.962,E2 -28409.962} C_VEL
LIN {X 0,Y 111.968,Z 643.462,A -85,B 0,C 180,E1 -28404.414,E2 -28404.414} C_VEL
LIN {X 0,Y 111.925,Z 643.475,A -85,B 0,C 180,E1 -28398.674,E2 -28398.674} C_VEL
LIN {X 0,Y 111.928,Z 643.473,A -85,B 0,C 180,E1 -28391.329,E2 -28391.329} C_VEL
LIN {X 0,Y 111.988,Z 643.458,A -85,B 0,C 180,E1 -28384.257,E2 -28384.257} C_VEL
LIN {X 0,Y 111.992,Z 643.467,A -85,B 0,C 180,E1 -28378.885,E2 -28378.885} C_VEL
LIN {X 0,Y 112.036,Z 643.457,A -85,B 0,C 180,E1 -28372.031,E2 -28372.031} C_VEL
LIN {X 0,Y 112.18,Z 643.444,A -85,B 0,C 180,E1 -28368.191,E2 -28368.191} C_VEL
LIN {X 0,Y 112.398,Z 643.416,A -85,B 0,C 180,E1 -28360.774,E2 -28360.774} C_VEL
LIN {X 0,Y 112.821,Z 643.359,A -85,B 0,C 180,E1 -28356.624,E2 -28356.624} C_VEL
LIN {X 0,Y 113.216,Z 643.316,A -85,B 0,C 180,E1 -28349.999,E2 -28349.999} C_VEL
LIN {X 0,Y 112.72,Z 643.373,A -85,B 0,C 180,E1 -28342.86,E2 -28342.86} C_VEL
LIN {X 0,Y 112.226,Z 643.428,A -85,B 0,C 180,E1 -28335.542,E2 -28335.542} C_VEL
LIN {X 0,Y 112.146,Z 643.447,A -85,B 0,C 180,E1 -28329.529,E2 -28329.529} C_VEL
LIN {X 0,Y 111.968,Z 643.464,A -85,B 0,C 180,E1 -28324.029,E2 -28324.029} C_VEL
LIN {X 0,Y 111.922,Z 643.476,A -85,B 0,C 180,E1 -28319.955,E2 -28319.955} C_VEL
LIN {X 0,Y 111.956,Z 643.465,A -85,B 0,C 180,E1 -28314.42,E2 -28314.42} C_VEL
LIN {X 0,Y 111.899,Z 643.477,A -85,B 0,C 180,E1 -28308.688,E2 -28308.688} C_VEL
LIN {X 0,Y 111.941,Z 643.472,A -85,B 0,C 180,E1 -28303.494,E2 -28303.494} C_VEL
LIN {X 0,Y 112.216,Z 643.43,A -85,B 0,C 180,E1 -28295.761,E2 -28295.761} C_VEL
LIN {X 0,Y 113.422,Z 643.284,A -85,B 0,C 180,E1 -28287.278,E2 -28287.278} C_VEL
LIN {X 0,Y 115.967,Z 669.799,A -85,B 0,C 180,E1 -28284.498,E2 -28284.498} C_VEL
LIN {X 0,Y 115.769,Z 731.434,A -85,B 0,C 180,E1 -28277.108,E2 -28277.108} C_VEL
LIN {X 0,Y 115.659,Z 746.758,A -85,B 0,C 180,E1 -28274.965,E2 -28274.965} C_VEL
LIN {X 0,Y 115.469,Z 759.729,A -85,B 0,C 180,E1 -28272.358,E2 -28272.358} C_VEL
LIN {X 0,Y 115.501,Z 770.553,A -85,B 0,C 180,E1 -28269.599,E2 -28269.599} C_VEL
LIN {X 0,Y 115.592,Z 780.2,A -85,B 0,C 180,E1 -28266.523,E2 -28266.523} C_VEL
LIN {X 0,Y 115.649,Z 788.167,A -85,B 0,C 180,E1 -28263.471,E2 -28263.471} C_VEL
LIN {X 0,Y 115.728,Z 795.754,A -85,B 0,C 180,E1 -28259.999,E2 -28259.999} C_VEL
LIN {X 0,Y 116.46,Z 806.53,A -85,B 0,C 180,E1 -28253.957,E2 -28253.957} C_VEL
LIN {X 0,Y 118.231,Z 814.165,A -85,B 0,C 180,E1 -28248.898,E2 -28248.898} C_VEL
LIN {X 0,Y 121.645,Z 821.802,A -85,B 0,C 180,E1 -28243.266,E2 -28243.266} C_VEL
LIN {X 0,Y 125.761,Z 827.469,A -85,B 0,C 180,E1 -28238.774,E2 -28238.774} C_VEL
LIN {X 0,Y 132.946,Z 833.721,A -85,B 0,C 180,E1 -28233.393,E2 -28233.393} C_VEL
LIN {X 0,Y 139.237,Z 837.626,A -85,B 0,C 180,E1 -28229.797,E2 -28229.797} C_VEL
LIN {X 0,Y 148.905,Z 841.622,A -85,B 0,C 180,E1 -28225.633,E2 -28225.633} C_VEL
LIN {X 0,Y 154.189,Z 843.209,A -85,B 0,C 180,E1 -28223.803,E2 -28223.803} C_VEL
LIN {X 0,Y 159.932,Z 844.436,A -85,B 0,C 180,E1 -28222.031,E2 -28222.031} C_VEL
LIN {X 0,Y 163.669,Z 845.161,A -85,B 0,C 180,E1 -28220.385,E2 -28220.385} C_VEL
LIN {X 0,Y 152.848,Z 843.419,A -85,B 0,C 180,E1 -28217.158,E2 -28217.158} C_VEL
LIN {X 0,Y 142.951,Z 840.561,A -85,B 0,C 180,E1 -28213.314,E2 -28213.314} C_VEL
LIN {X 0,Y 136.447,Z 837.749,A -85,B 0,C 180,E1 -28209.918,E2 -28209.918} C_VEL
LIN {X 0,Y 128.89,Z 832.829,A -85,B 0,C 180,E1 -28204.794,E2 -28204.794} C_VEL
LIN {X 0,Y 124.257,Z 828.407,A -85,B 0,C 180,E1 -28200.487,E2 -28200.487} C_VEL
LIN {X 0,Y 119.857,Z 821.13,A -85,B 0,C 180,E1 -28194.148,E2 -28194.148} C_VEL
LIN {X 0,Y 117.945,Z 814.84,A -85,B 0,C 180,E1 -28189.063,E2 -28189.063} C_VEL
LIN {X 0,Y 117.48,Z 805.854,A -85,B 0,C 180,E1 -28182.819,E2 -28182.819} C_VEL
LIN {X 0,Y 117.723,Z 800.19,A -85,B 0,C 180,E1 -28179.418,E2 -28179.418} C_VEL
LIN {X 0,Y 117.599,Z 794.649,A -85,B 0,C 180,E1 -28176.842,E2 -28176.842} C_VEL
LIN {X 0,Y 117.098,Z 786.985,A -85,B 0,C 180,E1 -28173.859,E2 -28173.859} C_VEL
LIN {X 0,Y 116.762,Z 779.224,A -85,B 0,C 180,E1 -28171.29,E2 -28171.29} C_VEL
LIN {X 0,Y 116.587,Z 773.409,A -85,B 0,C 180,E1 -28169.619,E2 -28169.619} C_VEL
LIN {X 0,Y 116.214,Z 769.905,A -85,B 0,C 180,E1 -28168.754,E2 -28168.754} C_VEL
LIN {X 0,Y 114.912,Z 764.457,A -85,B 0,C 180,E1 -28167.784,E2 -28167.784} C_VEL
LIN {X 0,Y 110.49,Z 749.688,A -85,B 0,C 180,E1 -28166.036,E2 -28166.036} C_VEL
LIN {X 0,Y 109.891,Z 743.7,A -85,B 0,C 180,E1 -28165.261,E2 -28165.261} C_VEL
LIN {X 0,Y 109.504,Z 715.81,A -85,B 0,C 180,E1 -28161.61,E2 -28161.61} C_VEL
LIN {X 0,Y 109.199,Z 689.472,A -85,B 0,C 180,E1 -28158.291,E2 -28158.291} C_VEL
LIN {X 0,Y 106.095,Z 656.941,A -85,B 0,C 180,E1 -28154.688,E2 -28154.688} C_VEL
LIN {X 0,Y 105.55,Z 644.266,A -85,B 0,C 180,E1 -28153.123,E2 -28153.123} C_VEL
LIN {X 0,Y 105.182,Z 644.317,A -85,B 0,C 180,E1 -28146.45,E2 -28146.45} C_VEL
LIN {X 0,Y 105.088,Z 644.317,A -85,B 0,C 180,E1 -28140.055,E2 -28140.055} C_VEL
LIN {X 0,Y 104.873,Z 644.35,A -85,B 0,C 180,E1 -28133.051,E2 -28133.051} C_VEL
LIN {X 0,Y 104.824,Z 644.36,A -85,B 0,C 180,E1 -28127.311,E2 -28127.311} C_VEL
LIN {X 0,Y 104.822,Z 644.35,A -85,B 0,C 180,E1 -28121.931,E2 -28121.931} C_VEL
LIN {X 0,Y 104.876,Z 644.353,A -85,B 0,C 180,E1 -28116.732,E2 -28116.732} C_VEL
LIN {X 0,Y 104.885,Z 644.347,A -85,B 0,C 180,E1 -28109.755,E2 -28109.755} C_VEL
LIN {X 0,Y 105.026,Z 644.326,A -85,B 0,C 180,E1 -28100.984,E2 -28100.984} C_VEL
LIN {X 0,Y 105.081,Z 644.326,A -85,B 0,C 180,E1 -28095.465,E2 -28095.465} C_VEL
LIN {X 0,Y 105.763,Z 644.243,A -85,B 0,C 180,E1 -28086.583,E2 -28086.583} C_VEL
LIN {X 0,Y 106.181,Z 644.187,A -85,B 0,C 180,E1 -28080.001,E2 -28080.001} C_VEL
LIN {X 0,Y 105.752,Z 644.235,A -85,B 0,C 180,E1 -28073.469,E2 -28073.469} C_VEL
LIN {X 0,Y 105.098,Z 644.319,A -85,B 0,C 180,E1 -28064.54,E2 -28064.54} C_VEL
LIN {X 0,Y 105.043,Z 644.332,A -85,B 0,C 180,E1 -28058.993,E2 -28058.993} C_VEL
LIN {X 0,Y 104.895,Z 644.349,A -85,B 0,C 180,E1 -28050.236,E2 -28050.236} C_VEL
LIN {X 0,Y 104.874,Z 644.344,A -85,B 0,C 180,E1 -28043.053,E2 -28043.053} C_VEL
LIN {X 0,Y 104.868,Z 644.353,A -85,B 0,C 180,E1 -28037.283,E2 -28037.283} C_VEL
LIN {X 0,Y 104.87,Z 644.349,A -85,B 0,C 180,E1 -28031.906,E2 -28031.906} C_VEL
LIN {X 0,Y 104.889,Z 644.35,A -85,B 0,C 180,E1 -28026.743,E2 -28026.743} C_VEL
LIN {X 0,Y 104.917,Z 644.349,A -85,B 0,C 180,E1 -28019.787,E2 -28019.787} C_VEL
LIN {X 0,Y 105.07,Z 644.328,A -85,B 0,C 180,E1 -28011.049,E2 -28011.049} C_VEL
LIN {X 0,Y 105.129,Z 644.313,A -85,B 0,C 180,E1 -28005.456,E2 -28005.456} C_VEL
LIN {X 0,Y 105.762,Z 644.237,A -85,B 0,C 180,E1 -27996.586,E2 -27996.586} C_VEL
LIN {X 0,Y 106.18,Z 644.192,A -85,B 0,C 180,E1 -27989.999,E2 -27989.999} C_VEL
LIN {X 0,Y 105.602,Z 644.26,A -85,B 0,C 180,E1 -27982.376,E2 -27982.376} C_VEL
LIN {X 0,Y 105.13,Z 644.313,A -85,B 0,C 180,E1 -27974.543,E2 -27974.543} C_VEL
LIN {X 0,Y 105.066,Z 644.329,A -85,B 0,C 180,E1 -27968.957,E2 -27968.957} C_VEL
LIN {X 0,Y 104.883,Z 644.354,A -85,B 0,C 180,E1 -27960.245,E2 -27960.245} C_VEL
LIN {X 0,Y 104.869,Z 644.352,A -85,B 0,C 180,E1 -27953.048,E2 -27953.048} C_VEL
LIN {X 0,Y 104.853,Z 644.348,A -85,B 0,C 180,E1 -27947.29,E2 -27947.29} C_VEL
LIN {X 0,Y 104.88,Z 644.354,A -85,B 0,C 180,E1 -27941.899,E2 -27941.899} C_VEL
LIN {X 0,Y 105.066,Z 644.32,A -85,B 0,C 180,E1 -27936.868,E2 -27936.868} C_VEL
LIN {X 0,Y 106.585,Z 644.135,A -85,B 0,C 180,E1 -27926.375,E2 -27926.375} C_VEL
LIN {X 0,Y 109.102,Z 670.503,A -85,B 0,C 180,E1 -27923.454,E2 -27923.454} C_VEL
LIN {X 0,Y 109.22,Z 730.503,A -85,B 0,C 180,E1 -27915.806,E2 -27915.806} C_VEL
LIN {X 0,Y 109.219,Z 746.322,A -85,B 0,C 180,E1 -27913.443,E2 -27913.443} C_VEL
LIN {X 0,Y 109.147,Z 759.372,A -85,B 0,C 180,E1 -27910.631,E2 -27910.631} C_VEL
LIN {X 0,Y 109.307,Z 769.742,A -85,B 0,C 180,E1 -27907.825,E2 -27907.825} C_VEL
LIN {X 0,Y 109.541,Z 780.632,A -85,B 0,C 180,E1 -27904.124,E2 -27904.124} C_VEL
LIN {X 0,Y 109.645,Z 788.363,A -85,B 0,C 180,E1 -27900.914,E2 -27900.914} C_VEL
LIN {X 0,Y 109.863,Z 797.331,A -85,B 0,C 180,E1 -27896.343,E2 -27896.343} C_VEL
LIN {X 0,Y 111.07,Z 806.215,A -85,B 0,C 180,E1 -27890.928,E2 -27890.928} C_VEL
LIN {X 0,Y 113.799,Z 815.006,A -85,B 0,C 180,E1 -27884.834,E2 -27884.834} C_VEL
LIN {X 0,Y 116.653,Z 820.538,A -85,B 0,C 180,E1 -27880.715,E2 -27880.715} C_VEL
LIN {X 0,Y 122.996,Z 827.99,A -85,B 0,C 180,E1 -27874.715,E2 -27874.715} C_VEL
LIN {X 0,Y 128.87,Z 832.835,A -85,B 0,C 180,E1 -27870.713,E2 -27870.713} C_VEL
LIN {X 0,Y 138.002,Z 837.993,A -85,B 0,C 180,E1 -27866.06,E2 -27866.06} C_VEL
LIN {X 0,Y 148.44,Z 841.965,A -85,B 0,C 180,E1 -27862.161,E2 -27862.161} C_VEL
LIN {X 0,Y 151.969,Z 842.977,A -85,B 0,C 180,E1 -27861.063,E2 -27861.063} C_VEL
LIN {X 0,Y 150.422,Z 842.678,A -85,B 0,C 180,E1 -27859.845,E2 -27859.845} C_VEL
LIN {X 0,Y 142.977,Z 840.65,A -85,B 0,C 180,E1 -27857.295,E2 -27857.295} C_VEL
LIN {X 0,Y 135.729,Z 837.956,A -85,B 0,C 180,E1 -27854.162,E2 -27854.162} C_VEL
LIN {X 0,Y 127.846,Z 833.704,A -85,B 0,C 180,E1 -27849.758,E2 -27849.758} C_VEL
LIN {X 0,Y 120.187,Z 827.282,A -85,B 0,C 180,E1 -27843.619,E2 -27843.619} C_VEL
LIN {X 0,Y 115.53,Z 821.01,A -85,B 0,C 180,E1 -27838.027,E2 -27838.027} C_VEL
LIN {X 0,Y 112.647,Z 813.57,A -85,B 0,C 180,E1 -27831.907,E2 -27831.907} C_VEL
LIN {X 0,Y 111.545,Z 805.328,A -85,B 0,C 180,E1 -27825.776,E2 -27825.776} C_VEL
LIN {X 0,Y 111.726,Z 799.136,A -85,B 0,C 180,E1 -27821.757,E2 -27821.757} C_VEL
LIN {X 0,Y 111.727,Z 793.798,A -85,B 0,C 180,E1 -27819.018,E2 -27819.018} C_VEL
LIN {X 0,Y 111.154,Z 786.154,A -85,B 0,C 180,E1 -27815.878,E2 -27815.878} C_VEL
LIN {X 0,Y 110.635,Z 777.01,A -85,B 0,C 180,E1 -27812.722,E2 -27812.722} C_VEL
LIN {X 0,Y 110.292,Z 767.509,A -85,B 0,C 180,E1 -27810.001,E2 -27810.001} C_VEL
LIN {X 0,Y 110.105,Z 757.824,A -85,B 0,C 180,E1 -27807.722,E2 -27807.722} C_VEL
LIN {X 0,Y 109.929,Z 747.061,A -85,B 0,C 180,E1 -27805.776,E2 -27805.776} C_VEL
LIN {X 0,Y 109.891,Z 743.7,A -85,B 0,C 180,E1 -27805.261,E2 -27805.261} C_VEL
LIN {X 0,Y 109.287,Z 737.99,A -85,B 0,C 180,E1 -27804.563,E2 -27804.563} C_VEL
LIN {X 0,Y 106.599,Z 728.532,A -85,B 0,C 180,E1 -27803.93,E2 -27803.93} C_VEL
LIN {X 0,Y 103.75,Z 719.034,A -85,B 0,C 180,E1 -27803.363,E2 -27803.363} C_VEL
LIN {X 0,Y 102.924,Z 713.251,A -85,B 0,C 180,E1 -27802.762,E2 -27802.762} C_VEL
LIN {X 0,Y 102.487,Z 689.372,A -85,B 0,C 180,E1 -27799.541,E2 -27799.541} C_VEL
LIN {X 0,Y 99.334,Z 657.927,A -85,B 0,C 180,E1 -27795.881,E2 -27795.881} C_VEL
LIN {X 0,Y 98.681,Z 645.124,A -85,B 0,C 180,E1 -27794.142,E2 -27794.142} C_VEL
LIN {X 0,Y 98.075,Z 645.201,A -85,B 0,C 180,E1 -27784.628,E2 -27784.628} C_VEL
LIN {X 0,Y 97.963,Z 645.209,A -85,B 0,C 180,E1 -27779.096,E2 -27779.096} C_VEL
LIN {X 0,Y 97.75,Z 645.231,A -85,B 0,C 180,E1 -27772.022,E2 -27772.022} C_VEL
LIN {X 0,Y 97.72,Z 645.242,A -85,B 0,C 180,E1 -27764.211,E2 -27764.211} C_VEL
LIN {X 0,Y 97.748,Z 645.24,A -85,B 0,C 180,E1 -27757.98,E2 -27757.98} C_VEL
LIN {X 0,Y 97.824,Z 645.225,A -85,B 0,C 180,E1 -27750.082,E2 -27750.082} C_VEL
LIN {X 0,Y 97.985,Z 645.203,A -85,B 0,C 180,E1 -27740.943,E2 -27740.943} C_VEL
LIN {X 0,Y 98.146,Z 645.182,A -85,B 0,C 180,E1 -27732.364,E2 -27732.364} C_VEL
LIN {X 0,Y 98.697,Z 645.123,A -85,B 0,C 180,E1 -27726.509,E2 -27726.509} C_VEL
LIN {X 0,Y 99.122,Z 645.066,A -85,B 0,C 180,E1 -27720.001,E2 -27720.001} C_VEL
LIN {X 0,Y 98.689,Z 645.114,A -85,B 0,C 180,E1 -27713.53,E2 -27713.53} C_VEL
LIN {X 0,Y 98.155,Z 645.191,A -85,B 0,C 180,E1 -27707.64,E2 -27707.64} C_VEL
LIN {X 0,Y 98.003,Z 645.209,A -85,B 0,C 180,E1 -27699.063,E2 -27699.063} C_VEL
LIN {X 0,Y 97.834,Z 645.229,A -85,B 0,C 180,E1 -27689.925,E2 -27689.925} C_VEL
LIN {X 0,Y 97.762,Z 645.232,A -85,B 0,C 180,E1 -27682.01,E2 -27682.01} C_VEL
LIN {X 0,Y 97.778,Z 645.228,A -85,B 0,C 180,E1 -27674.247,E2 -27674.247} C_VEL
LIN {X 0,Y 97.769,Z 645.239,A -85,B 0,C 180,E1 -27667.997,E2 -27667.997} C_VEL
LIN {X 0,Y 97.857,Z 645.228,A -85,B 0,C 180,E1 -27660.069,E2 -27660.069} C_VEL
LIN {X 0,Y 98.033,Z 645.205,A -85,B 0,C 180,E1 -27650.931,E2 -27650.931} C_VEL
LIN {X 0,Y 98.177,Z 645.183,A -85,B 0,C 180,E1 -27642.358,E2 -27642.358} C_VEL
LIN {X 0,Y 98.697,Z 645.117,A -85,B 0,C 180,E1 -27636.516,E2 -27636.516} C_VEL
LIN {X 0,Y 99.121,Z 645.072,A -85,B 0,C 180,E1 -27629.999,E2 -27629.999} C_VEL
LIN {X 0,Y 98.697,Z 645.117,A -85,B 0,C 180,E1 -27623.482,E2 -27623.482} C_VEL
LIN {X 0,Y 98.178,Z 645.183,A -85,B 0,C 180,E1 -27617.64,E2 -27617.64} C_VEL
LIN {X 0,Y 98.028,Z 645.205,A -85,B 0,C 180,E1 -27609.067,E2 -27609.067} C_VEL
LIN {X 0,Y 97.823,Z 645.232,A -85,B 0,C 180,E1 -27599.918,E2 -27599.918} C_VEL
LIN {X 0,Y 97.754,Z 645.241,A -85,B 0,C 180,E1 -27592.015,E2 -27592.015} C_VEL
LIN {X 0,Y 97.779,Z 645.232,A -85,B 0,C 180,E1 -27584.244,E2 -27584.244} C_VEL
LIN {X 0,Y 97.914,Z 645.214,A -85,B 0,C 180,E1 -27578.102,E2 -27578.102} C_VEL
LIN {X 0,Y 98.72,Z 645.122,A -85,B 0,C 180,E1 -27569.778,E2 -27569.778} C_VEL
LIN {X 0,Y 99.744,Z 644.99,A -85,B 0,C 180,E1 -27565.334,E2 -27565.334} C_VEL
LIN {X 0,Y 102.288,Z 669.86,A -85,B 0,C 180,E1 -27562.438,E2 -27562.438} C_VEL
LIN {X 0,Y 102.814,Z 727.932,A -85,B 0,C 180,E1 -27554.446,E2 -27554.446} C_VEL
LIN {X 0,Y 102.975,Z 744.087,A -85,B 0,C 180,E1 -27551.943,E2 -27551.943} C_VEL
LIN {X 0,Y 102.954,Z 758.457,A -85,B 0,C 180,E1 -27548.804,E2 -27548.804} C_VEL
LIN {X 0,Y 103.261,Z 770.355,A -85,B 0,C 180,E1 -27545.35,E2 -27545.35} C_VEL
LIN {X 0,Y 103.56,Z 779.803,A -85,B 0,C 180,E1 -27541.937,E2 -27541.937} C_VEL
LIN {X 0,Y 103.832,Z 788.393,A -85,B 0,C 180,E1 -27538.066,E2 -27538.066} C_VEL
LIN {X 0,Y 104.579,Z 798.535,A -85,B 0,C 180,E1 -27532.301,E2 -27532.301} C_VEL
LIN {X 0,Y 106.402,Z 807.185,A -85,B 0,C 180,E1 -27526.678,E2 -27526.678} C_VEL
LIN {X 0,Y 109.342,Z 814.579,A -85,B 0,C 180,E1 -27521.318,E2 -27521.318} C_VEL
LIN {X 0,Y 113.548,Z 821.081,A -85,B 0,C 180,E1 -27516.36,E2 -27516.36} C_VEL
LIN {X 0,Y 120.093,Z 827.873,A -85,B 0,C 180,E1 -27511.032,E2 -27511.032} C_VEL
LIN {X 0,Y 127.435,Z 833.2,A -85,B 0,C 180,E1 -27506.656,E2 -27506.656} C_VEL
LIN {X 0,Y 137.399,Z 838.34,A -85,B 0,C 180,E1 -27502.283,E2 -27502.283} C_VEL
LIN {X 0,Y 140.901,Z 839.735,A -85,B 0,C 180,E1 -27501.055,E2 -27501.055} C_VEL
LIN {X 0,Y 139.99,Z 839.488,A -85,B 0,C 180,E1 -27499.956,E2 -27499.956} C_VEL
LIN {X 0,Y 130.964,Z 835.832,A -85,B 0,C 180,E1 -27496.223,E2 -27496.223} C_VEL
LIN {X 0,Y 124.177,Z 832.152,A -85,B 0,C 180,E1 -27492.602,E2 -27492.602} C_VEL
LIN {X 0,Y 116.492,Z 826.087,A -85,B 0,C 180,E1 -27486.963,E2 -27486.963} C_VEL
LIN {X 0,Y 111.841,Z 820.732,A -85,B 0,C 180,E1 -27482.165,E2 -27482.165} C_VEL
LIN {X 0,Y 108.048,Z 813.487,A -85,B 0,C 180,E1 -27475.95,E2 -27475.95} C_VEL
LIN {X 0,Y 106.104,Z 804.864,A -85,B 0,C 180,E1 -27469.274,E2 -27469.274} C_VEL
LIN {X 0,Y 105.882,Z 797.903,A -85,B 0,C 180,E1 -27464.364,E2 -27464.364} C_VEL
LIN {X 0,Y 105.963,Z 792.892,A -85,B 0,C 180,E1 -27461.439,E2 -27461.439} C_VEL
LIN {X 0,Y 105.373,Z 785.33,A -85,B 0,C 180,E1 -27458.121,E2 -27458.121} C_VEL
LIN {X 0,Y 104.684,Z 776.133,A -85,B 0,C 180,E1 -27454.798,E2 -27454.798} C_VEL
LIN {X 0,Y 104.232,Z 766.587,A -85,B 0,C 180,E1 -27451.926,E2 -27451.926} C_VEL
LIN {X 0,Y 103.944,Z 756.813,A -85,B 0,C 180,E1 -27449.518,E2 -27449.518} C_VEL
LIN {X 0,Y 103.679,Z 746.825,A -85,B 0,C 180,E1 -27447.581,E2 -27447.581} C_VEL
LIN {X 0,Y 103.136,Z 721.629,A -85,B 0,C 180,E1 -27443.909,E2 -27443.909} C_VEL
LIN {X 0,Y 102.924,Z 713.251,A -85,B 0,C 180,E1 -27442.762,E2 -27442.762} C_VEL
LIN {X 0,Y 102.16,Z 707.493,A -85,B 0,C 180,E1 -27442.135,E2 -27442.135} C_VEL
LIN {X 0,Y 95.843,Z 686.687,A -85,B 0,C 180,E1 -27440.709,E2 -27440.709} C_VEL
LIN {X 0,Y 95.092,Z 682.829,A -85,B 0,C 180,E1 -27440.325,E2 -27440.325} C_VEL
LIN {X 0,Y 92.326,Z 653.366,A -85,B 0,C 180,E1 -27436.566,E2 -27436.566} C_VEL
LIN {X 0,Y 91.962,Z 645.959,A -85,B 0,C 180,E1 -27435.528,E2 -27435.528} C_VEL
LIN {X 0,Y 91.059,Z 646.074,A -85,B 0,C 180,E1 -27427.381,E2 -27427.381} C_VEL
LIN {X 0,Y 90.958,Z 646.08,A -85,B 0,C 180,E1 -27422.482,E2 -27422.482} C_VEL
LIN {X 0,Y 90.795,Z 646.107,A -85,B 0,C 180,E1 -27417.316,E2 -27417.316} C_VEL
LIN {X 0,Y 90.693,Z 646.109,A -85,B 0,C 180,E1 -27410.565,E2 -27410.565} C_VEL
LIN {X 0,Y 90.673,Z 646.119,A -85,B 0,C 180,E1 -27404.048,E2 -27404.048} C_VEL
LIN {X 0,Y 90.693,Z 646.118,A -85,B 0,C 180,E1 -27398.161,E2 -27398.161} C_VEL
LIN {X 0,Y 90.692,Z 646.11,A -85,B 0,C 180,E1 -27391.837,E2 -27391.837} C_VEL
LIN {X 0,Y 90.691,Z 646.121,A -85,B 0,C 180,E1 -27387.608,E2 -27387.608} C_VEL
LIN {X 0,Y 90.843,Z 646.091,A -85,B 0,C 180,E1 -27382.295,E2 -27382.295} C_VEL
LIN {X 0,Y 90.874,Z 646.098,A -85,B 0,C 180,E1 -27377.959,E2 -27377.959} C_VEL
LIN {X 0,Y 91.346,Z 646.037,A -85,B 0,C 180,E1 -27368.823,E2 -27368.823} C_VEL
LIN {X 0,Y 91.715,Z 645.987,A -85,B 0,C 180,E1 -27364.381,E2 -27364.381} C_VEL
LIN {X 0,Y 92.062,Z 645.945,A -85,B 0,C 180,E1 -27360.001,E2 -27360.001} C_VEL
LIN {X 0,Y 91.628,Z 645.994,A -85,B 0,C 180,E1 -27353.599,E2 -27353.599} C_VEL
LIN {X 0,Y 91.031,Z 646.078,A -85,B 0,C 180,E1 -27346.655,E2 -27346.655} C_VEL
LIN {X 0,Y 90.891,Z 646.085,A -85,B 0,C 180,E1 -27342.047,E2 -27342.047} C_VEL
LIN {X 0,Y 90.825,Z 646.103,A -85,B 0,C 180,E1 -27337.321,E2 -27337.321} C_VEL
LIN {X 0,Y 90.698,Z 646.11,A -85,B 0,C 180,E1 -27332.397,E2 -27332.397} C_VEL
LIN {X 0,Y 90.673,Z 646.122,A -85,B 0,C 180,E1 -27327.268,E2 -27327.268} C_VEL
LIN {X 0,Y 90.711,Z 646.116,A -85,B 0,C 180,E1 -27320.548,E2 -27320.548} C_VEL
LIN {X 0,Y 90.722,Z 646.106,A -85,B 0,C 180,E1 -27314.016,E2 -27314.016} C_VEL
LIN {X 0,Y 90.717,Z 646.118,A -85,B 0,C 180,E1 -27308.147,E2 -27308.147} C_VEL
LIN {X 0,Y 90.734,Z 646.11,A -85,B 0,C 180,E1 -27301.882,E2 -27301.882} C_VEL
LIN {X 0,Y 90.716,Z 646.116,A -85,B 0,C 180,E1 -27297.598,E2 -27297.598} C_VEL
LIN {X 0,Y 90.885,Z 646.091,A -85,B 0,C 180,E1 -27292.361,E2 -27292.361} C_VEL
LIN {X 0,Y 90.925,Z 646.09,A -85,B 0,C 180,E1 -27287.946,E2 -27287.946} C_VEL
LIN {X 0,Y 91.054,Z 646.067,A -85,B 0,C 180,E1 -27283.342,E2 -27283.342} C_VEL
LIN {X 0,Y 91.645,Z 645.994,A -85,B 0,C 180,E1 -27276.503,E2 -27276.503} C_VEL
LIN {X 0,Y 92.062,Z 645.951,A -85,B 0,C 180,E1 -27269.999,E2 -27269.999} C_VEL
LIN {X 0,Y 91.645,Z 645.994,A -85,B 0,C 180,E1 -27263.495,E2 -27263.495} C_VEL
LIN {X 0,Y 91.054,Z 646.067,A -85,B 0,C 180,E1 -27256.656,E2 -27256.656} C_VEL
LIN {X 0,Y 90.923,Z 646.09,A -85,B 0,C 180,E1 -27252.051,E2 -27252.051} C_VEL
LIN {X 0,Y 90.861,Z 646.093,A -85,B 0,C 180,E1 -27247.328,E2 -27247.328} C_VEL
LIN {X 0,Y 90.696,Z 646.118,A -85,B 0,C 180,E1 -27242.394,E2 -27242.394} C_VEL
LIN {X 0,Y 90.667,Z 646.116,A -85,B 0,C 180,E1 -27237.262,E2 -27237.262} C_VEL
LIN {X 0,Y 90.701,Z 646.12,A -85,B 0,C 180,E1 -27230.555,E2 -27230.555} C_VEL
LIN {X 0,Y 90.727,Z 646.111,A -85,B 0,C 180,E1 -27224.012,E2 -27224.012} C_VEL
LIN {X 0,Y 90.865,Z 646.091,A -85,B 0,C 180,E1 -27218.073,E2 -27218.073} C_VEL
LIN {X 0,Y 92.151,Z 645.931,A -85,B 0,C 180,E1 -27207.132,E2 -27207.132} C_VEL
LIN {X 0,Y 92.996,Z 645.833,A -85,B 0,C 180,E1 -27204.067,E2 -27204.067} C_VEL
LIN {X 0,Y 95.575,Z 670.687,A -85,B 0,C 180,E1 -27200.952,E2 -27200.952} C_VEL
LIN {X 0,Y 96.547,Z 729.222,A -85,B 0,C 180,E1 -27192.304,E2 -27192.304} C_VEL
LIN {X 0,Y 96.796,Z 744.422,A -85,B 0,C 180,E1 -27189.763,E2 -27189.763} C_VEL
LIN {X 0,Y 96.892,Z 757.486,A -85,B 0,C 180,E1 -27186.745,E2 -27186.745} C_VEL
LIN {X 0,Y 97.341,Z 769.484,A -85,B 0,C 180,E1 -27183.092,E2 -27183.092} C_VEL
LIN {X 0,Y 97.897,Z 779.879,A -85,B 0,C 180,E1 -27178.974,E2 -27178.974} C_VEL
LIN {X 0,Y 98.269,Z 788.088,A -85,B 0,C 180,E1 -27174.887,E2 -27174.887} C_VEL
LIN {X 0,Y 99.429,Z 798.153,A -85,B 0,C 180,E1 -27168.828,E2 -27168.828} C_VEL
LIN {X 0,Y 101.806,Z 806.671,A -85,B 0,C 180,E1 -27162.997,E2 -27162.997} C_VEL
LIN {X 0,Y 106.132,Z 815.147,A -85,B 0,C 180,E1 -27156.671,E2 -27156.671} C_VEL
LIN {X 0,Y 112,Z 822.47,A -85,B 0,C 180,E1 -27151.113,E2 -27151.113} C_VEL
LIN {X 0,Y 119.479,Z 828.842,A -85,B 0,C 180,E1 -27146.155,E2 -27146.155} C_VEL
LIN {X 0,Y 126.695,Z 833.545,A -85,B 0,C 180,E1 -27142.544,E2 -27142.544} C_VEL
LIN {X 0,Y 130.315,Z 835.422,A -85,B 0,C 180,E1 -27141.049,E2 -27141.049} C_VEL
LIN {X 0,Y 128.827,Z 834.808,A -85,B 0,C 180,E1 -27139.57,E2 -27139.57} C_VEL
LIN {X 0,Y 122.193,Z 831.306,A -85,B 0,C 180,E1 -27136.304,E2 -27136.304} C_VEL
LIN {X 0,Y 115.202,Z 826.561,A -85,B 0,C 180,E1 -27131.977,E2 -27131.977} C_VEL
LIN {X 0,Y 108.84,Z 820.398,A -85,B 0,C 180,E1 -27126.534,E2 -27126.534} C_VEL
LIN {X 0,Y 104.074,Z 813.209,A -85,B 0,C 180,E1 -27120.317,E2 -27120.317} C_VEL
LIN {X 0,Y 101.43,Z 806.149,A -85,B 0,C 180,E1 -27114.479,E2 -27114.479} C_VEL
LIN {X 0,Y 100.37,Z 796.423,A -85,B 0,C 180,E1 -27107.254,E2 -27107.254} C_VEL
LIN {X 0,Y 100.27,Z 789.885,A -85,B 0,C 180,E1 -27103.123,E2 -27103.123} C_VEL
LIN {X 0,Y 99.493,Z 782.462,A -85,B 0,C 180,E1 -27099.78,E2 -27099.78} C_VEL
LIN {X 0,Y 98.589,Z 771.768,A -85,B 0,C 180,E1 -27095.914,E2 -27095.914} C_VEL
LIN {X 0,Y 98.011,Z 758.215,A -85,B 0,C 180,E1 -27092.092,E2 -27092.092} C_VEL
LIN {X 0,Y 97.595,Z 747.103,A -85,B 0,C 180,E1 -27089.744,E2 -27089.744} C_VEL
LIN {X 0,Y 96.895,Z 723.896,A -85,B 0,C 180,E1 -27086.115,E2 -27086.115} C_VEL
LIN {X 0,Y 95.846,Z 689.044,A -85,B 0,C 180,E1 -27081.067,E2 -27081.067} C_VEL
LIN {X 0,Y 95.092,Z 682.829,A -85,B 0,C 180,E1 -27080.325,E2 -27080.325} C_VEL
LIN {X 0,Y 93.713,Z 677.129,A -85,B 0,C 180,E1 -27079.817,E2 -27079.817} C_VEL
LIN {X 0,Y 86.602,Z 658.731,A -85,B 0,C 180,E1 -27078.742,E2 -27078.742} C_VEL
LIN {X 0,Y 85.632,Z 653.031,A -85,B 0,C 180,E1 -27078.061,E2 -27078.061} C_VEL
LIN {X 0,Y 85.253,Z 646.794,A -85,B 0,C 180,E1 -27077.047,E2 -27077.047} C_VEL
LIN {X 0,Y 83.893,Z 646.969,A -85,B 0,C 180,E1 -27065.326,E2 -27065.326} C_VEL
LIN {X 0,Y 83.775,Z 646.972,A -85,B 0,C 180,E1 -27059.891,E2 -27059.891} C_VEL
LIN {X 0,Y 83.61,Z 647,A -85,B 0,C 180,E1 -27054.097,E2 -27054.097} C_VEL
LIN {X 0,Y 83.577,Z 647.005,A -85,B 0,C 180,E1 -27047.898,E2 -27047.898} C_VEL
LIN {X 0,Y 83.584,Z 646.994,A -85,B 0,C 180,E1 -27041.045,E2 -27041.045} C_VEL
LIN {X 0,Y 83.596,Z 646.996,A -85,B 0,C 180,E1 -27033.084,E2 -27033.084} C_VEL
LIN {X 0,Y 83.654,Z 646.995,A -85,B 0,C 180,E1 -27024.751,E2 -27024.751} C_VEL
LIN {X 0,Y 83.762,Z 646.979,A -85,B 0,C 180,E1 -27019.543,E2 -27019.543} C_VEL
LIN {X 0,Y 83.888,Z 646.963,A -85,B 0,C 180,E1 -27014.508,E2 -27014.508} C_VEL
LIN {X 0,Y 84.58,Z 646.882,A -85,B 0,C 180,E1 -27006.402,E2 -27006.402} C_VEL
LIN {X 0,Y 85.003,Z 646.825,A -85,B 0,C 180,E1 -27000.002,E2 -27000.002} C_VEL
LIN {X 0,Y 84.573,Z 646.873,A -85,B 0,C 180,E1 -26993.639,E2 -26993.639} C_VEL
LIN {X 0,Y 83.899,Z 646.963,A -85,B 0,C 180,E1 -26985.497,E2 -26985.497} C_VEL
LIN {X 0,Y 83.737,Z 646.986,A -85,B 0,C 180,E1 -26976.942,E2 -26976.942} C_VEL
LIN {X 0,Y 83.595,Z 647.003,A -85,B 0,C 180,E1 -26969.82,E2 -26969.82} C_VEL
LIN {X 0,Y 83.578,Z 646.996,A -85,B 0,C 180,E1 -26964.082,E2 -26964.082} C_VEL
LIN {X 0,Y 83.603,Z 647.003,A -85,B 0,C 180,E1 -26957.916,E2 -26957.916} C_VEL
LIN {X 0,Y 83.609,Z 647,A -85,B 0,C 180,E1 -26951.066,E2 -26951.066} C_VEL
LIN {X 0,Y 83.632,Z 646.99,A -85,B 0,C 180,E1 -26943.123,E2 -26943.123} C_VEL
LIN {X 0,Y 83.699,Z 646.981,A -85,B 0,C 180,E1 -26934.735,E2 -26934.735} C_VEL
LIN {X 0,Y 83.804,Z 646.979,A -85,B 0,C 180,E1 -26929.53,E2 -26929.53} C_VEL
LIN {X 0,Y 83.923,Z 646.952,A -85,B 0,C 180,E1 -26924.5,E2 -26924.5} C_VEL
LIN {X 0,Y 84.579,Z 646.874,A -85,B 0,C 180,E1 -26916.408,E2 -26916.408} C_VEL
LIN {X 0,Y 85.002,Z 646.83,A -85,B 0,C 180,E1 -26909.999,E2 -26909.999} C_VEL
LIN {X 0,Y 84.579,Z 646.874,A -85,B 0,C 180,E1 -26903.59,E2 -26903.59} C_VEL
LIN {X 0,Y 83.922,Z 646.952,A -85,B 0,C 180,E1 -26895.498,E2 -26895.498} C_VEL
LIN {X 0,Y 83.775,Z 646.973,A -85,B 0,C 180,E1 -26886.879,E2 -26886.879} C_VEL
LIN {X 0,Y 83.59,Z 647.004,A -85,B 0,C 180,E1 -26879.815,E2 -26879.815} C_VEL
LIN {X 0,Y 83.571,Z 647.001,A -85,B 0,C 180,E1 -26874.076,E2 -26874.076} C_VEL
LIN {X 0,Y 83.59,Z 646.998,A -85,B 0,C 180,E1 -26867.904,E2 -26867.904} C_VEL
LIN {X 0,Y 83.69,Z 646.993,A -85,B 0,C 180,E1 -26861.125,E2 -26861.125} C_VEL
LIN {X 0,Y 84.553,Z 646.886,A -85,B 0,C 180,E1 -26849.803,E2 -26849.803} C_VEL
LIN {X 0,Y 86.38,Z 646.854,A -85,B 0,C 180,E1 -26842.494,E2 -26842.494} C_VEL
LIN {X 0,Y 88.96,Z 670.078,A -85,B 0,C 180,E1 -26839.438,E2 -26839.438} C_VEL
LIN {X 0,Y 90.451,Z 730.444,A -85,B 0,C 180,E1 -26829.892,E2 -26829.892} C_VEL
LIN {X 0,Y 90.801,Z 745.133,A -85,B 0,C 180,E1 -26827.2,E2 -26827.2} C_VEL
LIN {X 0,Y 91.23,Z 759.301,A -85,B 0,C 180,E1 -26823.511,E2 -26823.511} C_VEL
LIN {X 0,Y 91.817,Z 769.666,A -85,B 0,C 180,E1 -26819.999,E2 -26819.999} C_VEL
LIN {X 0,Y 92.502,Z 779.769,A -85,B 0,C 180,E1 -26815.656,E2 -26815.656} C_VEL
LIN {X 0,Y 93.225,Z 789.467,A -85,B 0,C 180,E1 -26810.266,E2 -26810.266} C_VEL
LIN {X 0,Y 95.17,Z 799.047,A -85,B 0,C 180,E1 -26803.977,E2 -26803.977} C_VEL
LIN {X 0,Y 99.034,Z 808.541,A -85,B 0,C 180,E1 -26797.106,E2 -26797.106} C_VEL
LIN {X 0,Y 103.694,Z 815.694,A -85,B 0,C 180,E1 -26791.78,E2 -26791.78} C_VEL
LIN {X 0,Y 110.13,Z 822.464,A -85,B 0,C 180,E1 -26786.722,E2 -26786.722} C_VEL
LIN {X 0,Y 118.816,Z 829.192,A -85,B 0,C 180,E1 -26781.756,E2 -26781.756} C_VEL
LIN {X 0,Y 121.341,Z 830.795,A -85,B 0,C 180,E1 -26780.581,E2 -26780.581} C_VEL
LIN {X 0,Y 117.809,Z 828.769,A -85,B 0,C 180,E1 -26778.683,E2 -26778.683} C_VEL
LIN {X 0,Y 108.43,Z 821.856,A -85,B 0,C 180,E1 -26772.711,E2 -26772.711} C_VEL
LIN {X 0,Y 101.459,Z 813.95,A -85,B 0,C 180,E1 -26765.932,E2 -26765.932} C_VEL
LIN {X 0,Y 96.879,Z 804.573,A -85,B 0,C 180,E1 -26758.035,E2 -26758.035} C_VEL
LIN {X 0,Y 95.291,Z 797.732,A -85,B 0,C 180,E1 -26752.566,E2 -26752.566} C_VEL
LIN {X 0,Y 94.933,Z 789.06,A -85,B 0,C 180,E1 -26746.424,E2 -26746.424} C_VEL
LIN {X 0,Y 94.429,Z 783.245,A -85,B 0,C 180,E1 -26743.405,E2 -26743.405} C_VEL
LIN {X 0,Y 93.015,Z 771.295,A -85,B 0,C 180,E1 -26738.663,E2 -26738.663} C_VEL
LIN {X 0,Y 92.188,Z 758.935,A -85,B 0,C 180,E1 -26734.861,E2 -26734.861} C_VEL
LIN {X 0,Y 91.639,Z 747.315,A -85,B 0,C 180,E1 -26732.191,E2 -26732.191} C_VEL
LIN {X 0,Y 90.767,Z 725.65,A -85,B 0,C 180,E1 -26728.558,E2 -26728.558} C_VEL
LIN {X 0,Y 89.407,Z 689.196,A -85,B 0,C 180,E1 -26722.899,E2 -26722.899} C_VEL
LIN {X 0,Y 85.781,Z 655.865,A -85,B 0,C 180,E1 -26718.486,E2 -26718.486} C_VEL
LIN {X 0,Y 85.632,Z 653.031,A -85,B 0,C 180,E1 -26718.061,E2 -26718.061} C_VEL
LIN {X 0,Y 85.137,Z 650.84,A -85,B 0,C 180,E1 -26717.301,E2 -26717.301} C_VEL
LIN {X 0,Y 83.855,Z 648.871,A -85,B 0,C 180,E1 -26715.565,E2 -26715.565} C_VEL
LIN {X 0,Y 81.874,Z 647.659,A -85,B 0,C 180,E1 -26712.72,E2 -26712.72} C_VEL
LIN {X 0,Y 80.357,Z 647.4,A -85,B 0,C 180,E1 -26710.216,E2 -26710.216} C_VEL
LIN {X 0,Y 76.783,Z 647.855,A -85,B 0,C 180,E1 -26700.357,E2 -26700.357} C_VEL
LIN {X 0,Y 76.64,Z 647.869,A -85,B 0,C 180,E1 -26696.886,E2 -26696.886} C_VEL
LIN {X 0,Y 76.502,Z 647.877,A -85,B 0,C 180,E1 -26690.142,E2 -26690.142} C_VEL
LIN {X 0,Y 76.495,Z 647.881,A -85,B 0,C 180,E1 -26682.902,E2 -26682.902} C_VEL
LIN {X 0,Y 76.517,Z 647.883,A -85,B 0,C 180,E1 -26674.528,E2 -26674.528} C_VEL
LIN {X 0,Y 76.651,Z 647.864,A -85,B 0,C 180,E1 -26663.964,E2 -26663.964} C_VEL
LIN {X 0,Y 76.741,Z 647.857,A -85,B 0,C 180,E1 -26655.893,E2 -26655.893} C_VEL
LIN {X 0,Y 77.524,Z 647.761,A -85,B 0,C 180,E1 -26646.355,E2 -26646.355} C_VEL
LIN {X 0,Y 77.943,Z 647.704,A -85,B 0,C 180,E1 -26640.002,E2 -26640.002} C_VEL
LIN {X 0,Y 77.506,Z 647.753,A -85,B 0,C 180,E1 -26633.768,E2 -26633.768} C_VEL
LIN {X 0,Y 76.75,Z 647.847,A -85,B 0,C 180,E1 -26624.112,E2 -26624.112} C_VEL
LIN {X 0,Y 76.654,Z 647.866,A -85,B 0,C 180,E1 -26616.03,E2 -26616.03} C_VEL
LIN {X 0,Y 76.524,Z 647.879,A -85,B 0,C 180,E1 -26605.465,E2 -26605.465} C_VEL
LIN {X 0,Y 76.517,Z 647.885,A -85,B 0,C 180,E1 -26597.08,E2 -26597.08} C_VEL
LIN {X 0,Y 76.514,Z 647.886,A -85,B 0,C 180,E1 -26589.851,E2 -26589.851} C_VEL
LIN {X 0,Y 76.589,Z 647.867,A -85,B 0,C 180,E1 -26583.279,E2 -26583.279} C_VEL
LIN {X 0,Y 76.695,Z 647.853,A -85,B 0,C 180,E1 -26574.041,E2 -26574.041} C_VEL
LIN {X 0,Y 76.796,Z 647.842,A -85,B 0,C 180,E1 -26565.879,E2 -26565.879} C_VEL
LIN {X 0,Y 77.573,Z 647.743,A -85,B 0,C 180,E1 -26555.18,E2 -26555.18} C_VEL
LIN {X 0,Y 77.943,Z 647.709,A -85,B 0,C 180,E1 -26549.999,E2 -26549.999} C_VEL
LIN {X 0,Y 77.522,Z 647.752,A -85,B 0,C 180,E1 -26543.645,E2 -26543.645} C_VEL
LIN {X 0,Y 76.796,Z 647.842,A -85,B 0,C 180,E1 -26534.119,E2 -26534.119} C_VEL
LIN {X 0,Y 76.684,Z 647.854,A -85,B 0,C 180,E1 -26525.977,E2 -26525.977} C_VEL
LIN {X 0,Y 76.518,Z 647.875,A -85,B 0,C 180,E1 -26515.47,E2 -26515.47} C_VEL
LIN {X 0,Y 76.515,Z 647.876,A -85,B 0,C 180,E1 -26507.08,E2 -26507.08} C_VEL
LIN {X 0,Y 76.626,Z 647.871,A -85,B 0,C 180,E1 -26499.78,E2 -26499.78} C_VEL
LIN {X 0,Y 77.073,Z 647.816,A -85,B 0,C 180,E1 -26493.042,E2 -26493.042} C_VEL
LIN {X 0,Y 79.784,Z 647.478,A -85,B 0,C 180,E1 -26480.725,E2 -26480.725} C_VEL
LIN {X 0,Y 82.395,Z 670.279,A -85,B 0,C 180,E1 -26477.527,E2 -26477.527} C_VEL
LIN {X 0,Y 84.231,Z 722.624,A -85,B 0,C 180,E1 -26468.582,E2 -26468.582} C_VEL
LIN {X 0,Y 85.025,Z 741.376,A -85,B 0,C 180,E1 -26465.126,E2 -26465.126} C_VEL
LIN {X 0,Y 85.354,Z 751.672,A -85,B 0,C 180,E1 -26462.585,E2 -26462.585} C_VEL
LIN {X 0,Y 85.942,Z 761.579,A -85,B 0,C 180,E1 -26459.561,E2 -26459.561} C_VEL
LIN {X 0,Y 86.686,Z 771.122,A -85,B 0,C 180,E1 -26455.944,E2 -26455.944} C_VEL
LIN {X 0,Y 87.36,Z 779.551,A -85,B 0,C 180,E1 -26451.933,E2 -26451.933} C_VEL
LIN {X 0,Y 88.507,Z 788.862,A -85,B 0,C 180,E1 -26446.264,E2 -26446.264} C_VEL
LIN {X 0,Y 91.663,Z 799.782,A -85,B 0,C 180,E1 -26438.716,E2 -26438.716} C_VEL
LIN {X 0,Y 95.704,Z 807.852,A -85,B 0,C 180,E1 -26432.777,E2 -26432.777} C_VEL
LIN {X 0,Y 102.122,Z 816.034,A -85,B 0,C 180,E1 -26426.72,E2 -26426.72} C_VEL
LIN {X 0,Y 108.76,Z 822.329,A -85,B 0,C 180,E1 -26422.277,E2 -26422.277} C_VEL
LIN {X 0,Y 111.164,Z 824.203,A -85,B 0,C 180,E1 -26420.941,E2 -26420.941} C_VEL
LIN {X 0,Y 110.56,Z 823.828,A -85,B 0,C 180,E1 -26419.487,E2 -26419.487} C_VEL
LIN {X 0,Y 101.913,Z 816.508,A -85,B 0,C 180,E1 -26413.418,E2 -26413.418} C_VEL
LIN {X 0,Y 95.164,Z 807.922,A -85,B 0,C 180,E1 -26406.075,E2 -26406.075} C_VEL
LIN {X 0,Y 90.976,Z 797.612,A -85,B 0,C 180,E1 -26397.514,E2 -26397.514} C_VEL
LIN {X 0,Y 89.772,Z 788.649,A -85,B 0,C 180,E1 -26390.559,E2 -26390.559} C_VEL
LIN {X 0,Y 89.707,Z 785.099,A -85,B 0,C 180,E1 -26388.2,E2 -26388.2} C_VEL
LIN {X 0,Y 88.861,Z 778.652,A -85,B 0,C 180,E1 -26384.992,E2 -26384.992} C_VEL
LIN {X 0,Y 87.632,Z 769.112,A -85,B 0,C 180,E1 -26381.236,E2 -26381.236} C_VEL
LIN {X 0,Y 86.636,Z 757.529,A -85,B 0,C 180,E1 -26377.55,E2 -26377.55} C_VEL
LIN {X 0,Y 85.912,Z 746.367,A -85,B 0,C 180,E1 -26374.824,E2 -26374.824} C_VEL
LIN {X 0,Y 84.654,Z 722.813,A -85,B 0,C 180,E1 -26370.591,E2 -26370.591} C_VEL
LIN {X 0,Y 82.979,Z 688.692,A -85,B 0,C 180,E1 -26364.931,E2 -26364.931} C_VEL
LIN {X 0,Y 79.185,Z 655.617,A -85,B 0,C 180,E1 -26360.293,E2 -26360.293} C_VEL
LIN {X 0,Y 78.655,Z 647.616,A -85,B 0,C 180,E1 -26358.935,E2 -26358.935} C_VEL
LIN {X 0,Y 76.862,Z 647.845,A -85,B 0,C 180,E1 -26345.69,E2 -26345.69} C_VEL
LIN {X 0,Y 76.64,Z 647.869,A -85,B 0,C 180,E1 -26336.886,E2 -26336.886} C_VEL
LIN {X 0,Y 76.431,Z 647.916,A -85,B 0,C 180,E1 -26333.969,E2 -26333.969} C_VEL
LIN {X 0,Y 75.09,Z 648.093,A -85,B 0,C 180,E1 -26329.626,E2 -26329.626} C_VEL
LIN {X 0,Y 71.709,Z 648.493,A -85,B 0,C 180,E1 -26322.21,E2 -26322.21} C_VEL
LIN {X 0,Y 69.606,Z 648.747,A -85,B 0,C 180,E1 -26315.747,E2 -26315.747} C_VEL
LIN {X 0,Y 69.308,Z 648.768,A -85,B 0,C 180,E1 -26312.365,E2 -26312.365} C_VEL
LIN {X 0,Y 69.622,Z 648.738,A -85,B 0,C 180,E1 -26303.732,E2 -26303.732} C_VEL
LIN {X 0,Y 69.623,Z 648.745,A -85,B 0,C 180,E1 -26297.568,E2 -26297.568} C_VEL
LIN {X 0,Y 70.52,Z 648.631,A -85,B 0,C 180,E1 -26285.702,E2 -26285.702} C_VEL
LIN {X 0,Y 70.863,Z 648.586,A -85,B 0,C 180,E1 -26280.002,E2 -26280.002} C_VEL
LIN {X 0,Y 70.445,Z 648.632,A -85,B 0,C 180,E1 -26273.875,E2 -26273.875} C_VEL
LIN {X 0,Y 69.631,Z 648.732,A -85,B 0,C 180,E1 -26262.437,E2 -26262.437} C_VEL
LIN {X 0,Y 69.537,Z 648.748,A -85,B 0,C 180,E1 -26255.032,E2 -26255.032} C_VEL
LIN {X 0,Y 69.388,Z 648.773,A -85,B 0,C 180,E1 -26249.689,E2 -26249.689} C_VEL
LIN {X 0,Y 69.394,Z 648.762,A -85,B 0,C 180,E1 -26242.729,E2 -26242.729} C_VEL
LIN {X 0,Y 69.428,Z 648.759,A -85,B 0,C 180,E1 -26234.926,E2 -26234.926} C_VEL
LIN {X 0,Y 69.443,Z 648.761,A -85,B 0,C 180,E1 -26226.207,E2 -26226.207} C_VEL
LIN {X 0,Y 69.414,Z 648.77,A -85,B 0,C 180,E1 -26220.3,E2 -26220.3} C_VEL
LIN {X 0,Y 69.665,Z 648.728,A -85,B 0,C 180,E1 -26213.713,E2 -26213.713} C_VEL
LIN {X 0,Y 69.671,Z 648.736,A -85,B 0,C 180,E1 -26207.553,E2 -26207.553} C_VEL
LIN {X 0,Y 70.519,Z 648.622,A -85,B 0,C 180,E1 -26195.699,E2 -26195.699} C_VEL
LIN {X 0,Y 70.864,Z 648.591,A -85,B 0,C 180,E1 -26189.999,E2 -26189.999} C_VEL
LIN {X 0,Y 70.457,Z 648.631,A -85,B 0,C 180,E1 -26183.779,E2 -26183.779} C_VEL
LIN {X 0,Y 69.668,Z 648.737,A -85,B 0,C 180,E1 -26172.444,E2 -26172.444} C_VEL
LIN {X 0,Y 69.561,Z 648.741,A -85,B 0,C 180,E1 -26164.987,E2 -26164.987} C_VEL
LIN {X 0,Y 69.39,Z 648.773,A -85,B 0,C 180,E1 -26159.686,E2 -26159.686} C_VEL
LIN {X 0,Y 69.389,Z 648.772,A -85,B 0,C 180,E1 -26152.722,E2 -26152.722} C_VEL
LIN {X 0,Y 69.465,Z 648.755,A -85,B 0,C 180,E1 -26144.895,E2 -26144.895} C_VEL
LIN {X 0,Y 69.701,Z 648.723,A -85,B 0,C 180,E1 -26136.49,E2 -26136.49} C_VEL
LIN {X 0,Y 73.317,Z 648.281,A -85,B 0,C 180,E1 -26118.548,E2 -26118.548} C_VEL
LIN {X 0,Y 76.062,Z 670.497,A -85,B 0,C 180,E1 -26115.18,E2 -26115.18} C_VEL
LIN {X 0,Y 78.838,Z 727.97,A -85,B 0,C 180,E1 -26104.579,E2 -26104.579} C_VEL
LIN {X 0,Y 79.578,Z 742.372,A -85,B 0,C 180,E1 -26101.637,E2 -26101.637} C_VEL
LIN {X 0,Y 80.199,Z 754.054,A -85,B 0,C 180,E1 -26098.434,E2 -26098.434} C_VEL
LIN {X 0,Y 81.034,Z 763.886,A -85,B 0,C 180,E1 -26095.04,E2 -26095.04} C_VEL
LIN {X 0,Y 81.771,Z 771.024,A -85,B 0,C 180,E1 -26091.997,E2 -26091.997} C_VEL
LIN {X 0,Y 82.682,Z 778.977,A -85,B 0,C 180,E1 -26087.771,E2 -26087.771} C_VEL
LIN {X 0,Y 84.786,Z 789.786,A -85,B 0,C 180,E1 -26080.702,E2 -26080.702} C_VEL
LIN {X 0,Y 88.228,Z 799.019,A -85,B 0,C 180,E1 -26074.109,E2 -26074.109} C_VEL
LIN {X 0,Y 94.058,Z 808.272,A -85,B 0,C 180,E1 -26067.248,E2 -26067.248} C_VEL
LIN {X 0,Y 101.41,Z 816.408,A -85,B 0,C 180,E1 -26061.563,E2 -26061.563} C_VEL
LIN {X 0,Y 103.019,Z 817.869,A -85,B 0,C 180,E1 -26060.574,E2 -26060.574} C_VEL
LIN {X 0,Y 101.851,Z 816.899,A -85,B 0,C 180,E1 -26059.157,E2 -26059.157} C_VEL
LIN {X 0,Y 94.635,Z 809.554,A -85,B 0,C 180,E1 -26053.209,E2 -26053.209} C_VEL
LIN {X 0,Y 89.258,Z 801.517,A -85,B 0,C 180,E1 -26046.357,E2 -26046.357} C_VEL
LIN {X 0,Y 85.722,Z 791.323,A -85,B 0,C 180,E1 -26037.892,E2 -26037.892} C_VEL
LIN {X 0,Y 84.626,Z 781.703,A -85,B 0,C 180,E1 -26030.598,E2 -26030.598} C_VEL
LIN {X 0,Y 83.74,Z 775.849,A -85,B 0,C 180,E1 -26027.742,E2 -26027.742} C_VEL
LIN {X 0,Y 82.444,Z 766.883,A -85,B 0,C 180,E1 -26024.139,E2 -26024.139} C_VEL
LIN {X 0,Y 81.307,Z 755.945,A -85,B 0,C 180,E1 -26020.549,E2 -26020.549} C_VEL
LIN {X 0,Y 80.453,Z 745.168,A -85,B 0,C 180,E1 -26017.819,E2 -26017.819} C_VEL
LIN {X 0,Y 78.711,Z 719.002,A -85,B 0,C 180,E1 -26012.896,E2 -26012.896} C_VEL
LIN {X 0,Y 76.817,Z 688.572,A -85,B 0,C 180,E1 -26007.47,E2 -26007.47} C_VEL
LIN {X 0,Y 72.787,Z 655.656,A -85,B 0,C 180,E1 -26002.571,E2 -26002.571} C_VEL
LIN {X 0,Y 72.223,Z 648.412,A -85,B 0,C 180,E1 -26001.285,E2 -26001.285} C_VEL
LIN {X 0,Y 69.757,Z 648.728,A -85,B 0,C 180,E1 -25984.654,E2 -25984.654} C_VEL
LIN {X 0,Y 69.408,Z 648.753,A -85,B 0,C 180,E1 -25976.96,E2 -25976.96} C_VEL
LIN {X 0,Y 69.437,Z 648.759,A -85,B 0,C 180,E1 -25972.755,E2 -25972.755} C_VEL
LIN {X 0,Y 69.403,Z 648.772,A -85,B 0,C 180,E1 -25964.95,E2 -25964.95} C_VEL
LIN {X 0,Y 69.402,Z 648.773,A -85,B 0,C 180,E1 -25956.159,E2 -25956.159} C_VEL
LIN {X 0,Y 69.308,Z 648.768,A -85,B 0,C 180,E1 -25952.365,E2 -25952.365} C_VEL
LIN {X 0,Y 69.068,Z 648.809,A -85,B 0,C 180,E1 -25949.119,E2 -25949.119} C_VEL
LIN {X 0,Y 67.927,Z 648.96,A -85,B 0,C 180,E1 -25944.26,E2 -25944.26} C_VEL
LIN {X 0,Y 65.196,Z 649.312,A -85,B 0,C 180,E1 -25935.926,E2 -25935.926} C_VEL
LIN {X 0,Y 63.399,Z 649.513,A -85,B 0,C 180,E1 -25925.089,E2 -25925.089} C_VEL
LIN {X 0,Y 63.782,Z 649.467,A -85,B 0,C 180,E1 -25920.002,E2 -25920.002} C_VEL
LIN {X 0,Y 63.325,Z 649.518,A -85,B 0,C 180,E1 -25913.652,E2 -25913.652} C_VEL
LIN {X 0,Y 62.713,Z 649.606,A -85,B 0,C 180,E1 -25907.094,E2 -25907.094} C_VEL
LIN {X 0,Y 62.495,Z 649.628,A -85,B 0,C 180,E1 -25900.354,E2 -25900.354} C_VEL
LIN {X 0,Y 62.399,Z 649.632,A -85,B 0,C 180,E1 -25893.322,E2 -25893.322} C_VEL
LIN {X 0,Y 62.299,Z 649.651,A -85,B 0,C 180,E1 -25885.797,E2 -25885.797} C_VEL
LIN {X 0,Y 62.243,Z 649.663,A -85,B 0,C 180,E1 -25877.533,E2 -25877.533} C_VEL
LIN {X 0,Y 62.324,Z 649.654,A -85,B 0,C 180,E1 -25868.125,E2 -25868.125} C_VEL
LIN {X 0,Y 62.327,Z 649.642,A -85,B 0,C 180,E1 -25864.187,E2 -25864.187} C_VEL
LIN {X 0,Y 62.439,Z 649.632,A -85,B 0,C 180,E1 -25856.181,E2 -25856.181} C_VEL
LIN {X 0,Y 62.535,Z 649.628,A -85,B 0,C 180,E1 -25849.633,E2 -25849.633} C_VEL
LIN {X 0,Y 62.734,Z 649.594,A -85,B 0,C 180,E1 -25842.902,E2 -25842.902} C_VEL
